   1:L PR[91] R[100]mm/sec CNT100;
   1:  PR[GP1:91,1] = PR[GP1:90,1] + -38.837;
   1:  PR[GP1:91,2] = PR[GP1:90,2] + -4.762;
   1:L PR[91] R[100]mm/sec CNT100;
   1:  PR[GP1:91,1] = PR[GP1:90,1] + -38.715;
   1:  PR[GP1:91,2] = PR[GP1:90,2] + -5.232;
   1:L PR[91] R[100]mm/sec CNT100;
   1:  PR[GP1:91,1] = PR[GP1:90,1] + -37.344;
   1:  PR[GP1:91,2] = PR[GP1:90,2] + -8.646;
   1:L PR[91] R[100]mm/sec CNT100;
   1:  PR[GP1:91,1] = PR[GP1:90,1] + -37.044;
   1:  PR[GP1:91,2] = PR[GP1:90,2] + -9.321;
   1:L PR[91] R[100]mm/sec CNT100;
   1:  PR[GP1:91,1] = PR[GP1:90,1] + -35.099;
   1:  PR[GP1:91,2] = PR[GP1:90,2] + -12.020;
   1:L PR[91] R[100]mm/sec CNT100;
   1:  PR[GP1:91,1] = PR[GP1:90,1] + -34.536;
   1:  PR[GP1:91,2] = PR[GP1:90,2] + -12.886;
   1:L PR[91] R[100]mm/sec CNT100;
   1:  PR[GP1:91,1] = PR[GP1:90,1] + -33.800;
   1:  PR[GP1:91,2] = PR[GP1:90,2] + -13.678;
   1:L PR[91] R[100]mm/sec CNT100;
   1:  PR[GP1:91,1] = PR[GP1:90,1] + -31.666;
   1:  PR[GP1:91,2] = PR[GP1:90,2] + -15.488;
   1:L PR[91] R[100]mm/sec CNT100;
   1:  PR[GP1:91,1] = PR[GP1:90,1] + -30.501;
   1:  PR[GP1:91,2] = PR[GP1:90,2] + -16.399;
   1:L PR[91] R[100]mm/sec CNT100;
   1:  PR[GP1:91,1] = PR[GP1:90,1] + -28.778;
   1:  PR[GP1:91,2] = PR[GP1:90,2] + -17.354;
   1:L PR[91] R[100]mm/sec CNT100;
   1:  PR[GP1:91,1] = PR[GP1:90,1] + -27.068;
   1:  PR[GP1:91,2] = PR[GP1:90,2] + -18.219;
   1:L PR[91] R[100]mm/sec CNT100;
   1:  PR[GP1:91,1] = PR[GP1:90,1] + -24.860;
   1:  PR[GP1:91,2] = PR[GP1:90,2] + -19.021;
   1:L PR[91] R[100]mm/sec CNT100;
   1:  PR[GP1:91,1] = PR[GP1:90,1] + -23.856;
   1:  PR[GP1:91,2] = PR[GP1:90,2] + -19.262;
   1:L PR[91] R[100]mm/sec CNT100;
   1:  PR[GP1:91,1] = PR[GP1:90,1] + -21.199;
   1:  PR[GP1:91,2] = PR[GP1:90,2] + -19.791;
   1:L PR[91] R[100]mm/sec CNT100;
   1:  PR[GP1:91,1] = PR[GP1:90,1] + -17.823;
   1:  PR[GP1:91,2] = PR[GP1:90,2] + -19.955;
   1:L PR[91] R[100]mm/sec CNT100;
   1:  PR[GP1:91,1] = PR[GP1:90,1] + -14.672;
   1:  PR[GP1:91,2] = PR[GP1:90,2] + -19.637;
   1:L PR[91] R[100]mm/sec CNT100;
   1:  PR[GP1:91,1] = PR[GP1:90,1] + -14.261;
   1:  PR[GP1:91,2] = PR[GP1:90,2] + -19.580;
   1:L PR[91] R[100]mm/sec CNT100;
   1:  PR[GP1:91,1] = PR[GP1:90,1] + -11.329;
   1:  PR[GP1:91,2] = PR[GP1:90,2] + -18.822;
   1:L PR[91] R[100]mm/sec CNT100;
   1:  PR[GP1:91,1] = PR[GP1:90,1] + -7.839;
   1:  PR[GP1:91,2] = PR[GP1:90,2] + -17.303;
   1:L PR[91] R[100]mm/sec CNT100;
   1:  PR[GP1:91,1] = PR[GP1:90,1] + -5.607;
   1:  PR[GP1:91,2] = PR[GP1:90,2] + -15.876;
   1:L PR[91] R[100]mm/sec CNT100;
   1:  PR[GP1:91,1] = PR[GP1:90,1] + -5.328;
   1:  PR[GP1:91,2] = PR[GP1:90,2] + -15.675;
   1:L PR[91] R[100]mm/sec CNT100;
   1:  PR[GP1:91,1] = PR[GP1:90,1] + -4.271;
   1:  PR[GP1:91,2] = PR[GP1:90,2] + -14.749;
   1:L PR[91] R[100]mm/sec CNT100;
   1:  PR[GP1:91,1] = PR[GP1:90,1] + -3.185;
   1:  PR[GP1:91,2] = PR[GP1:90,2] + -13.771;
   1:L PR[91] R[100]mm/sec CNT100;
   1:  PR[GP1:91,1] = PR[GP1:90,1] + -2.156;
   1:  PR[GP1:91,2] = PR[GP1:90,2] + -12.565;
   1:L PR[91] R[100]mm/sec CNT100;
   1:  PR[GP1:91,1] = PR[GP1:90,1] + -1.829;
   1:  PR[GP1:91,2] = PR[GP1:90,2] + -12.302;
   1:L PR[91] R[100]mm/sec CNT100;
   1:  PR[GP1:91,1] = PR[GP1:90,1] + -0.550;
   1:  PR[GP1:91,2] = PR[GP1:90,2] + -11.397;
   1:L PR[91] R[100]mm/sec CNT100;
   1:  PR[GP1:91,1] = PR[GP1:90,1] + 0.193;
   1:  PR[GP1:91,2] = PR[GP1:90,2] + -11.661;
   1:L PR[91] R[100]mm/sec CNT100;
   1:  PR[GP1:91,1] = PR[GP1:90,1] + 1.144;
   1:L PR[91] R[100]mm/sec CNT100;
   1:  PR[GP1:91,1] = PR[GP1:90,1] + 1.657;
   1:  PR[GP1:91,2] = PR[GP1:90,2] + -12.081;
   1:L PR[91] R[100]mm/sec CNT100;
   1:  PR[GP1:91,1] = PR[GP1:90,1] + 2.294;
   1:  PR[GP1:91,2] = PR[GP1:90,2] + -12.534;
   1:L PR[91] R[100]mm/sec CNT100;
   1:  PR[GP1:91,1] = PR[GP1:90,1] + 3.356;
   1:  PR[GP1:91,2] = PR[GP1:90,2] + -13.783;
   1:L PR[91] R[100]mm/sec CNT100;
   1:  PR[GP1:91,1] = PR[GP1:90,1] + 4.441;
   1:  PR[GP1:91,2] = PR[GP1:90,2] + -14.761;
   1:L PR[91] R[100]mm/sec CNT100;
   1:  PR[GP1:91,1] = PR[GP1:90,1] + 5.471;
   1:  PR[GP1:91,2] = PR[GP1:90,2] + -15.664;
   1:L PR[91] R[100]mm/sec CNT100;
   1:  PR[GP1:91,1] = PR[GP1:90,1] + 7.593;
   1:  PR[GP1:91,2] = PR[GP1:90,2] + -17.023;
   1:L PR[91] R[100]mm/sec CNT100;
   1:  PR[GP1:91,1] = PR[GP1:90,1] + 8.015;
   1:  PR[GP1:91,2] = PR[GP1:90,2] + -17.314;
   1:L PR[91] R[100]mm/sec CNT100;
   1:  PR[GP1:91,1] = PR[GP1:90,1] + 11.478;
   1:  PR[GP1:91,2] = PR[GP1:90,2] + -18.817;
   1:L PR[91] R[100]mm/sec CNT100;
   1:  PR[GP1:91,1] = PR[GP1:90,1] + 14.391;
   1:  PR[GP1:91,2] = PR[GP1:90,2] + -19.572;
   1:L PR[91] R[100]mm/sec CNT100;
   1:  PR[GP1:91,1] = PR[GP1:90,1] + 17.974;
   1:  PR[GP1:91,2] = PR[GP1:90,2] + -19.955;
   1:L PR[91] R[100]mm/sec CNT100;
   1:  PR[GP1:91,1] = PR[GP1:90,1] + 21.307;
   1:  PR[GP1:91,2] = PR[GP1:90,2] + -19.796;
   1:L PR[91] R[100]mm/sec CNT100;
   1:  PR[GP1:91,1] = PR[GP1:90,1] + 21.648;
   1:  PR[GP1:91,2] = PR[GP1:90,2] + -19.716;
   1:L PR[91] R[100]mm/sec CNT100;
   1:  PR[GP1:91,1] = PR[GP1:90,1] + 25.016;
   1:  PR[GP1:91,2] = PR[GP1:90,2] + -19.018;
   1:L PR[91] R[100]mm/sec CNT100;
   1:  PR[GP1:91,1] = PR[GP1:90,1] + 27.213;
   1:  PR[GP1:91,2] = PR[GP1:90,2] + -18.224;
   1:L PR[91] R[100]mm/sec CNT100;
   1:  PR[GP1:91,1] = PR[GP1:90,1] + 28.922;
   1:  PR[GP1:91,2] = PR[GP1:90,2] + -17.361;
   1:L PR[91] R[100]mm/sec CNT100;
   1:  PR[GP1:91,1] = PR[GP1:90,1] + 30.618;
   1:  PR[GP1:91,2] = PR[GP1:90,2] + -16.426;
   1:L PR[91] R[100]mm/sec CNT100;
   1:  PR[GP1:91,1] = PR[GP1:90,1] + 32.732;
   1:  PR[GP1:91,2] = PR[GP1:90,2] + -14.641;
   1:L PR[91] R[100]mm/sec CNT100;
   1:  PR[GP1:91,1] = PR[GP1:90,1] + 33.954;
   1:  PR[GP1:91,2] = PR[GP1:90,2] + -13.677;
   1:L PR[91] R[100]mm/sec CNT100;
   1:  PR[GP1:91,1] = PR[GP1:90,1] + 34.702;
   1:  PR[GP1:91,2] = PR[GP1:90,2] + -12.874;
   1:L PR[91] R[100]mm/sec CNT100;
   1:  PR[GP1:91,1] = PR[GP1:90,1] + 36.691;
   1:  PR[GP1:91,2] = PR[GP1:90,2] + -10.095;
   1:L PR[91] R[100]mm/sec CNT100;
   1:  PR[GP1:91,1] = PR[GP1:90,1] + 37.186;
   1:  PR[GP1:91,2] = PR[GP1:90,2] + -9.346;
   1:L PR[91] R[100]mm/sec CNT100;
   1:  PR[GP1:91,1] = PR[GP1:90,1] + 37.499;
   1:  PR[GP1:91,2] = PR[GP1:90,2] + -8.654;
   1:L PR[91] R[100]mm/sec CNT100;
   1:  PR[GP1:91,1] = PR[GP1:90,1] + 38.869;
   1:  PR[GP1:91,2] = PR[GP1:90,2] + -5.258;
   1:L PR[91] R[100]mm/sec CNT100;
   1:  PR[GP1:91,1] = PR[GP1:90,1] + 38.999;
   1:  PR[GP1:91,2] = PR[GP1:90,2] + -4.762;
   1:L PR[91] R[100]mm/sec CNT100;
   1:  PR[GP1:91,1] = PR[GP1:90,1] + 39.503;
   1:  PR[GP1:91,2] = PR[GP1:90,2] + -0.771;
   1:L PR[91] R[100]mm/sec CNT100;
   1:  PR[GP1:91,1] = PR[GP1:90,1] + 39.538;
   1:  PR[GP1:91,2] = PR[GP1:90,2] + -0.345;
   1:L PR[91] R[100]mm/sec CNT100;
   1:  PR[GP1:91,1] = PR[GP1:90,1] + 39.040;
   1:  PR[GP1:91,2] = PR[GP1:90,2] + 3.557;
   1:L PR[91] R[100]mm/sec CNT100;
   1:  PR[GP1:91,1] = PR[GP1:90,1] + 38.991;
   1:  PR[GP1:91,2] = PR[GP1:90,2] + 4.171;
   1:L PR[91] R[100]mm/sec CNT100;
   1:  PR[GP1:91,1] = PR[GP1:90,1] + 38.869;
   1:  PR[GP1:91,2] = PR[GP1:90,2] + 4.635;
   1:L PR[91] R[100]mm/sec CNT100;
   1:  PR[GP1:91,1] = PR[GP1:90,1] + 37.498;
   1:  PR[GP1:91,2] = PR[GP1:90,2] + 8.032;
   1:L PR[91] R[100]mm/sec CNT100;
   1:  PR[GP1:91,1] = PR[GP1:90,1] + 37.197;
   1:  PR[GP1:91,2] = PR[GP1:90,2] + 8.698;
   1:L PR[91] R[100]mm/sec CNT100;
   1:  PR[GP1:91,1] = PR[GP1:90,1] + 35.251;
   1:  PR[GP1:91,2] = PR[GP1:90,2] + 11.401;
   1:L PR[91] R[100]mm/sec CNT100;
   1:  PR[GP1:91,1] = PR[GP1:90,1] + 34.679;
   1:  PR[GP1:91,2] = PR[GP1:90,2] + 12.274;
   1:L PR[91] R[100]mm/sec CNT100;
   1:  PR[GP1:91,1] = PR[GP1:90,1] + 33.934;
   1:  PR[GP1:91,2] = PR[GP1:90,2] + 13.074;
   1:L PR[91] R[100]mm/sec CNT100;
   1:  PR[GP1:91,1] = PR[GP1:90,1] + 31.800;
   1:  PR[GP1:91,2] = PR[GP1:90,2] + 14.887;
   1:L PR[91] R[100]mm/sec CNT100;
   1:  PR[GP1:91,1] = PR[GP1:90,1] + 30.641;
   1:  PR[GP1:91,2] = PR[GP1:90,2] + 15.790;
   1:L PR[91] R[100]mm/sec CNT100;
   1:  PR[GP1:91,1] = PR[GP1:90,1] + 28.920;
   1:  PR[GP1:91,2] = PR[GP1:90,2] + 16.738;
   1:L PR[91] R[100]mm/sec CNT100;
   1:  PR[GP1:91,1] = PR[GP1:90,1] + 27.211;
   1:  PR[GP1:91,2] = PR[GP1:90,2] + 17.600;
   1:L PR[91] R[100]mm/sec CNT100;
   1:  PR[GP1:91,1] = PR[GP1:90,1] + 24.993;
   1:  PR[GP1:91,2] = PR[GP1:90,2] + 18.402;
   1:L PR[91] R[100]mm/sec CNT100;
   1:  PR[GP1:91,1] = PR[GP1:90,1] + 23.992;
   1:  PR[GP1:91,2] = PR[GP1:90,2] + 18.642;
   1:L PR[91] R[100]mm/sec CNT100;
   1:  PR[GP1:91,1] = PR[GP1:90,1] + 21.332;
   1:  PR[GP1:91,2] = PR[GP1:90,2] + 19.171;
   1:L PR[91] R[100]mm/sec CNT100;
   1:  PR[GP1:91,1] = PR[GP1:90,1] + 17.971;
   1:  PR[GP1:91,2] = PR[GP1:90,2] + 19.331;
   1:L PR[91] R[100]mm/sec CNT100;
   1:  PR[GP1:91,1] = PR[GP1:90,1] + 14.829;
   1:  PR[GP1:91,2] = PR[GP1:90,2] + 19.012;
   1:L PR[91] R[100]mm/sec CNT100;
   1:  PR[GP1:91,1] = PR[GP1:90,1] + 14.418;
   1:  PR[GP1:91,2] = PR[GP1:90,2] + 18.955;
   1:L PR[91] R[100]mm/sec CNT100;
   1:  PR[GP1:91,1] = PR[GP1:90,1] + 11.487;
   1:  PR[GP1:91,2] = PR[GP1:90,2] + 18.196;
   1:L PR[91] R[100]mm/sec CNT100;
   1:  PR[GP1:91,1] = PR[GP1:90,1] + 8.920;
   1:  PR[GP1:91,2] = PR[GP1:90,2] + 17.072;
   1:L PR[91] R[100]mm/sec CNT100;
   1:  PR[GP1:91,1] = PR[GP1:90,1] + 8.012;
   1:  PR[GP1:91,2] = PR[GP1:90,2] + 16.693;
   1:L PR[91] R[100]mm/sec CNT100;
   1:  PR[GP1:91,1] = PR[GP1:90,1] + 5.789;
   1:  PR[GP1:91,2] = PR[GP1:90,2] + 15.274;
   1:L PR[91] R[100]mm/sec CNT100;
   1:  PR[GP1:91,1] = PR[GP1:90,1] + 5.612;
   1:  PR[GP1:91,2] = PR[GP1:90,2] + 15.152;
   1:L PR[91] R[100]mm/sec CNT100;
   1:  PR[GP1:91,1] = PR[GP1:90,1] + 5.268;
   1:  PR[GP1:91,2] = PR[GP1:90,2] + 14.879;
   1:L PR[91] R[100]mm/sec CNT100;
   1:  PR[GP1:91,1] = PR[GP1:90,1] + 3.427;
   1:  PR[GP1:91,2] = PR[GP1:90,2] + 13.229;
   1:L PR[91] R[100]mm/sec CNT100;
   1:  PR[GP1:91,1] = PR[GP1:90,1] + 2.786;
   1:  PR[GP1:91,2] = PR[GP1:90,2] + 12.556;
   1:L PR[91] R[100]mm/sec CNT100;
   1:  PR[GP1:91,1] = PR[GP1:90,1] + 2.184;
   1:  PR[GP1:91,2] = PR[GP1:90,2] + 11.814;
   1:L PR[91] R[100]mm/sec CNT100;
   1:  PR[GP1:91,1] = PR[GP1:90,1] + 1.393;
   1:  PR[GP1:91,2] = PR[GP1:90,2] + 11.254;
   1:L PR[91] R[100]mm/sec CNT100;
   1:  PR[GP1:91,1] = PR[GP1:90,1] + 0.820;
   1:  PR[GP1:91,2] = PR[GP1:90,2] + 10.940;
   1:L PR[91] R[100]mm/sec CNT100;
   1:  PR[GP1:91,1] = PR[GP1:90,1] + -0.635;
   1:L PR[91] R[100]mm/sec CNT100;
   1:  PR[91] = PR[90];
   1:  PR[GP1:91,1] = PR[GP1:90,1] + -1.462;
   1:  PR[GP1:91,2] = PR[GP1:90,2] + 11.634;
   1:  PR[GP1:91,3] = PR[GP1:90,3] + 27.145;
   1:L PR[91] R[100]mm/sec CNT100;
   1:  PR[GP1:91,1] = PR[GP1:90,1] + -1.730;
   1:  PR[GP1:91,2] = PR[GP1:90,2] + 11.982;
   1:L PR[91] R[100]mm/sec CNT100;
   1:  PR[GP1:91,1] = PR[GP1:90,1] + -1.967;
   1:  PR[GP1:91,2] = PR[GP1:90,2] + 12.206;
   1:L PR[91] R[100]mm/sec CNT100;
   1:  PR[GP1:91,1] = PR[GP1:90,1] + -2.120;
   1:  PR[GP1:91,2] = PR[GP1:90,2] + 12.316;
   1:L PR[91] R[100]mm/sec CNT100;
   1:  PR[GP1:91,1] = PR[GP1:90,1] + -2.321;
   1:  PR[GP1:91,2] = PR[GP1:90,2] + 12.557;
   1:L PR[91] R[100]mm/sec CNT100;
   1:  PR[GP1:91,1] = PR[GP1:90,1] + -3.063;
   1:  PR[GP1:91,2] = PR[GP1:90,2] + 13.334;
   1:L PR[91] R[100]mm/sec CNT100;
   1:  PR[GP1:91,1] = PR[GP1:90,1] + -4.810;
   1:  PR[GP1:91,2] = PR[GP1:90,2] + 14.896;
   1:L PR[91] R[100]mm/sec CNT100;
   1:  PR[GP1:91,1] = PR[GP1:90,1] + -5.202;
   1:  PR[GP1:91,2] = PR[GP1:90,2] + 15.206;
   1:L PR[91] R[100]mm/sec CNT100;
   1:  PR[GP1:91,1] = PR[GP1:90,1] + -7.585;
   1:  PR[GP1:91,2] = PR[GP1:90,2] + 16.743;
   1:L PR[91] R[100]mm/sec CNT100;
   1:  PR[GP1:91,1] = PR[GP1:90,1] + -10.209;
   1:  PR[GP1:91,2] = PR[GP1:90,2] + 17.890;
   1:L PR[91] R[100]mm/sec CNT100;
   1:  PR[GP1:91,1] = PR[GP1:90,1] + -11.131;
   1:  PR[GP1:91,2] = PR[GP1:90,2] + 18.276;
   1:L PR[91] R[100]mm/sec CNT100;
   1:  PR[GP1:91,1] = PR[GP1:90,1] + -13.916;
   1:  PR[GP1:91,2] = PR[GP1:90,2] + 18.996;
   1:L PR[91] R[100]mm/sec CNT100;
   1:  PR[GP1:91,1] = PR[GP1:90,1] + -17.278;
   1:  PR[GP1:91,2] = PR[GP1:90,2] + 19.346;
   1:L PR[91] R[100]mm/sec CNT100;
   1:  PR[GP1:91,1] = PR[GP1:90,1] + -17.623;
   1:  PR[GP1:91,2] = PR[GP1:90,2] + 19.393;
   1:L PR[91] R[100]mm/sec CNT100;
   1:  PR[GP1:91,1] = PR[GP1:90,1] + -20.933;
   1:  PR[GP1:91,2] = PR[GP1:90,2] + 19.218;
   1:L PR[91] R[100]mm/sec CNT100;
   1:  PR[GP1:91,1] = PR[GP1:90,1] + -24.493;
   1:  PR[GP1:91,2] = PR[GP1:90,2] + 18.487;
   1:L PR[91] R[100]mm/sec CNT100;
   1:  PR[GP1:91,1] = PR[GP1:90,1] + -27.043;
   1:  PR[GP1:91,2] = PR[GP1:90,2] + 17.561;
   1:L PR[91] R[100]mm/sec CNT100;
   1:  PR[GP1:91,1] = PR[GP1:90,1] + -28.228;
   1:  PR[GP1:91,2] = PR[GP1:90,2] + 16.962;
   1:L PR[91] R[100]mm/sec CNT100;
   1:  PR[GP1:91,1] = PR[GP1:90,1] + -30.293;
   1:  PR[GP1:91,2] = PR[GP1:90,2] + 15.817;
   1:L PR[91] R[100]mm/sec CNT100;
   1:  PR[GP1:91,1] = PR[GP1:90,1] + -31.942;
   1:  PR[GP1:91,2] = PR[GP1:90,2] + 14.426;
   1:L PR[91] R[100]mm/sec CNT100;
   1:  PR[GP1:91,1] = PR[GP1:90,1] + -33.508;
   1:  PR[GP1:91,2] = PR[GP1:90,2] + 13.187;
   1:L PR[91] R[100]mm/sec CNT100;
   1:  PR[GP1:91,1] = PR[GP1:90,1] + -34.483;
   1:  PR[GP1:91,2] = PR[GP1:90,2] + 12.138;
   1:L PR[91] R[100]mm/sec CNT100;
   1:  PR[GP1:91,1] = PR[GP1:90,1] + -36.170;
   1:  PR[GP1:91,2] = PR[GP1:90,2] + 9.783;
   1:L PR[91] R[100]mm/sec CNT100;
   1:  PR[GP1:91,1] = PR[GP1:90,1] + -36.854;
   1:  PR[GP1:91,2] = PR[GP1:90,2] + 8.743;
   1:L PR[91] R[100]mm/sec CNT100;
   1:  PR[GP1:91,1] = PR[GP1:90,1] + -37.298;
   1:  PR[GP1:91,2] = PR[GP1:90,2] + 7.745;
   1:L PR[91] R[100]mm/sec CNT100;
   1:  PR[GP1:91,1] = PR[GP1:90,1] + -38.498;
   1:  PR[GP1:91,2] = PR[GP1:90,2] + 4.758;
   1:L PR[91] R[100]mm/sec CNT100;
   1:  PR[GP1:91,1] = PR[GP1:90,1] + -38.706;
   1:  PR[GP1:91,2] = PR[GP1:90,2] + 3.951;
   1:L PR[91] R[100]mm/sec CNT100;
   1:  PR[GP1:91,1] = PR[GP1:90,1] + -39.150;
   1:  PR[GP1:91,2] = PR[GP1:90,2] + 0.453;
   1:L PR[91] R[100]mm/sec CNT100;
   1:  PR[GP1:91,1] = PR[GP1:90,1] + -39.207;
   1:  PR[GP1:91,2] = PR[GP1:90,2] + -0.277;
   1:L PR[91] R[100]mm/sec CNT100;
   1:  PR[GP1:91,1] = PR[GP1:90,1] + -38.768;
   1:  PR[GP1:91,2] = PR[GP1:90,2] + -3.707;
   1:L PR[91] R[100]mm/sec CNT100;
   1:  PR[GP1:91,1] = PR[GP1:90,1] + -38.698;
   1:  PR[GP1:91,2] = PR[GP1:90,2] + -4.608;
   1:L PR[91] R[100]mm/sec CNT100;
   1:  PR[GP1:91,1] = PR[GP1:90,1] + -38.498;
   1:  PR[GP1:91,2] = PR[GP1:90,2] + -5.382;
   1:L PR[91] R[100]mm/sec CNT100;
   1:  PR[GP1:91,1] = PR[GP1:90,1] + -37.298;
   1:  PR[GP1:91,2] = PR[GP1:90,2] + -8.369;
   1:L PR[91] R[100]mm/sec CNT100;
   1:  PR[GP1:91,1] = PR[GP1:90,1] + -36.866;
   1:  PR[GP1:91,2] = PR[GP1:90,2] + -9.338;
   1:L PR[91] R[100]mm/sec CNT100;
   1:  PR[GP1:91,1] = PR[GP1:90,1] + -35.185;
   1:  PR[GP1:91,2] = PR[GP1:90,2] + -11.672;
   1:L PR[91] R[100]mm/sec CNT100;
   1:  PR[GP1:91,1] = PR[GP1:90,1] + -34.460;
   1:  PR[GP1:91,2] = PR[GP1:90,2] + -12.786;
   1:L PR[91] R[100]mm/sec CNT100;
   1:  PR[GP1:91,1] = PR[GP1:90,1] + -33.492;
   1:  PR[GP1:91,2] = PR[GP1:90,2] + -13.829;
   1:L PR[91] R[100]mm/sec CNT100;
   1:  PR[GP1:91,1] = PR[GP1:90,1] + -31.736;
   1:  PR[GP1:91,2] = PR[GP1:90,2] + -15.318;
   1:L PR[91] R[100]mm/sec CNT100;
   1:  PR[GP1:91,1] = PR[GP1:90,1] + -30.316;
   1:  PR[GP1:91,2] = PR[GP1:90,2] + -16.428;
   1:L PR[91] R[100]mm/sec CNT100;
   1:  PR[GP1:91,1] = PR[GP1:90,1] + -28.228;
   1:  PR[GP1:91,2] = PR[GP1:90,2] + -17.586;
   1:L PR[91] R[100]mm/sec CNT100;
   1:  PR[GP1:91,1] = PR[GP1:90,1] + -27.043;
   1:  PR[GP1:91,2] = PR[GP1:90,2] + -18.185;
   1:L PR[91] R[100]mm/sec CNT100;
   1:  PR[GP1:91,1] = PR[GP1:90,1] + -24.471;
   1:  PR[GP1:91,2] = PR[GP1:90,2] + -19.119;
   1:L PR[91] R[100]mm/sec CNT100;
   1:  PR[GP1:91,1] = PR[GP1:90,1] + -24.001;
   1:  PR[GP1:91,2] = PR[GP1:90,2] + -19.232;
   1:L PR[91] R[100]mm/sec CNT100;
   1:  PR[GP1:91,1] = PR[GP1:90,1] + -21.022;
   1:  PR[GP1:91,2] = PR[GP1:90,2] + -19.832;
   1:L PR[91] R[100]mm/sec CNT100;
   1:  PR[GP1:91,1] = PR[GP1:90,1] + -17.593;
   1:  PR[GP1:91,2] = PR[GP1:90,2] + -20.018;
   1:L PR[91] R[100]mm/sec CNT100;
   1:  PR[GP1:91,1] = PR[GP1:90,1] + -14.573;
   1:  PR[GP1:91,2] = PR[GP1:90,2] + -19.714;
   1:L PR[91] R[100]mm/sec CNT100;
   1:  PR[GP1:91,1] = PR[GP1:90,1] + -13.934;
   1:  PR[GP1:91,2] = PR[GP1:90,2] + -19.625;
   1:L PR[91] R[100]mm/sec CNT100;
   1:  PR[GP1:91,1] = PR[GP1:90,1] + -11.131;
   1:  PR[GP1:91,2] = PR[GP1:90,2] + -18.900;
   1:L PR[91] R[100]mm/sec CNT100;
   1:  PR[GP1:91,1] = PR[GP1:90,1] + -7.545;
   1:  PR[GP1:91,2] = PR[GP1:90,2] + -17.342;
   1:L PR[91] R[100]mm/sec CNT100;
   1:  PR[GP1:91,1] = PR[GP1:90,1] + -5.422;
   1:  PR[GP1:91,2] = PR[GP1:90,2] + -15.984;
   1:L PR[91] R[100]mm/sec CNT100;
   1:  PR[GP1:91,1] = PR[GP1:90,1] + -5.084;
   1:  PR[GP1:91,2] = PR[GP1:90,2] + -15.740;
   1:L PR[91] R[100]mm/sec CNT100;
   1:  PR[GP1:91,1] = PR[GP1:90,1] + -3.847;
   1:  PR[GP1:91,2] = PR[GP1:90,2] + -14.658;
   1:L PR[91] R[100]mm/sec CNT100;
   1:  PR[GP1:91,1] = PR[GP1:90,1] + -2.979;
   1:  PR[GP1:91,2] = PR[GP1:90,2] + -13.875;
   1:L PR[91] R[100]mm/sec CNT100;
   1:  PR[GP1:91,1] = PR[GP1:90,1] + -2.138;
   1:  PR[GP1:91,2] = PR[GP1:90,2] + -12.889;
   1:L PR[91] R[100]mm/sec CNT100;
   1:  PR[GP1:91,1] = PR[GP1:90,1] + -1.752;
   1:  PR[GP1:91,2] = PR[GP1:90,2] + -12.580;
   1:L PR[91] R[100]mm/sec CNT100;
   1:  PR[GP1:91,1] = PR[GP1:90,1] + -0.525;
   1:  PR[GP1:91,2] = PR[GP1:90,2] + -11.712;
   1:L PR[91] R[100]mm/sec CNT100;
   1:  PR[GP1:91,1] = PR[GP1:90,1] + 0.316;
   1:  PR[GP1:91,2] = PR[GP1:90,2] + -12.011;
   1:L PR[91] R[100]mm/sec CNT100;
   1:  PR[GP1:91,1] = PR[GP1:90,1] + 1.168;
   1:L PR[91] R[100]mm/sec CNT100;
   1:  PR[GP1:91,1] = PR[GP1:90,1] + 1.737;
   1:  PR[GP1:91,2] = PR[GP1:90,2] + -12.477;
   1:L PR[91] R[100]mm/sec CNT100;
   1:  PR[GP1:91,1] = PR[GP1:90,1] + 2.275;
   1:  PR[GP1:91,2] = PR[GP1:90,2] + -12.859;
   1:L PR[91] R[100]mm/sec CNT100;
   1:  PR[GP1:91,1] = PR[GP1:90,1] + 3.148;
   1:  PR[GP1:91,2] = PR[GP1:90,2] + -13.886;
   1:L PR[91] R[100]mm/sec CNT100;
   1:  PR[GP1:91,1] = PR[GP1:90,1] + 4.015;
   1:  PR[GP1:91,2] = PR[GP1:90,2] + -14.668;
   1:L PR[91] R[100]mm/sec CNT100;
   1:  PR[GP1:91,1] = PR[GP1:90,1] + 5.225;
   1:  PR[GP1:91,2] = PR[GP1:90,2] + -15.728;
   1:L PR[91] R[100]mm/sec CNT100;
   1:  PR[GP1:91,1] = PR[GP1:90,1] + 7.196;
   1:  PR[GP1:91,2] = PR[GP1:90,2] + -16.991;
   1:L PR[91] R[100]mm/sec CNT100;
   1:  PR[GP1:91,1] = PR[GP1:90,1] + 7.721;
   1:  PR[GP1:91,2] = PR[GP1:90,2] + -17.352;
   1:L PR[91] R[100]mm/sec CNT100;
   1:  PR[GP1:91,1] = PR[GP1:90,1] + 11.280;
   1:  PR[GP1:91,2] = PR[GP1:90,2] + -18.895;
   1:L PR[91] R[100]mm/sec CNT100;
   1:  PR[GP1:91,1] = PR[GP1:90,1] + 14.063;
   1:  PR[GP1:91,2] = PR[GP1:90,2] + -19.617;
   1:L PR[91] R[100]mm/sec CNT100;
   1:  PR[GP1:91,1] = PR[GP1:90,1] + 17.421;
   1:  PR[GP1:91,2] = PR[GP1:90,2] + -19.969;
   1:L PR[91] R[100]mm/sec CNT100;
   1:  PR[GP1:91,1] = PR[GP1:90,1] + 17.768;
   1:  PR[GP1:91,2] = PR[GP1:90,2] + -20.017;
   1:L PR[91] R[100]mm/sec CNT100;
   1:  PR[GP1:91,1] = PR[GP1:90,1] + 21.063;
   1:  PR[GP1:91,2] = PR[GP1:90,2] + -19.846;
   1:L PR[91] R[100]mm/sec CNT100;
   1:  PR[GP1:91,1] = PR[GP1:90,1] + 24.625;
   1:  PR[GP1:91,2] = PR[GP1:90,2] + -19.116;
   1:L PR[91] R[100]mm/sec CNT100;
   1:  PR[GP1:91,1] = PR[GP1:90,1] + 27.186;
   1:  PR[GP1:91,2] = PR[GP1:90,2] + -18.191;
   1:L PR[91] R[100]mm/sec CNT100;
   1:  PR[GP1:91,1] = PR[GP1:90,1] + 28.369;
   1:  PR[GP1:91,2] = PR[GP1:90,2] + -17.594;
   1:L PR[91] R[100]mm/sec CNT100;
   1:  PR[GP1:91,1] = PR[GP1:90,1] + 30.431;
   1:  PR[GP1:91,2] = PR[GP1:90,2] + -16.457;
   1:L PR[91] R[100]mm/sec CNT100;
   1:  PR[GP1:91,1] = PR[GP1:90,1] + 32.078;
   1:  PR[GP1:91,2] = PR[GP1:90,2] + -15.066;
   1:L PR[91] R[100]mm/sec CNT100;
   1:  PR[GP1:91,1] = PR[GP1:90,1] + 33.640;
   1:  PR[GP1:91,2] = PR[GP1:90,2] + -13.833;
   1:L PR[91] R[100]mm/sec CNT100;
   1:  PR[GP1:91,1] = PR[GP1:90,1] + 34.622;
   1:  PR[GP1:91,2] = PR[GP1:90,2] + -12.778;
   1:L PR[91] R[100]mm/sec CNT100;
   1:  PR[GP1:91,1] = PR[GP1:90,1] + 36.310;
   1:  PR[GP1:91,2] = PR[GP1:90,2] + -10.421;
   1:L PR[91] R[100]mm/sec CNT100;
   1:  PR[GP1:91,1] = PR[GP1:90,1] + 37.008;
   1:  PR[GP1:91,2] = PR[GP1:90,2] + -9.366;
   1:L PR[91] R[100]mm/sec CNT100;
   1:  PR[GP1:91,1] = PR[GP1:90,1] + 37.451;
   1:  PR[GP1:91,2] = PR[GP1:90,2] + -8.384;
   1:L PR[91] R[100]mm/sec CNT100;
   1:  PR[GP1:91,1] = PR[GP1:90,1] + 38.650;
   1:  PR[GP1:91,2] = PR[GP1:90,2] + -5.412;
   1:L PR[91] R[100]mm/sec CNT100;
   1:  PR[GP1:91,1] = PR[GP1:90,1] + 38.859;
   1:  PR[GP1:91,2] = PR[GP1:90,2] + -4.616;
   1:L PR[91] R[100]mm/sec CNT100;
   1:  PR[GP1:91,1] = PR[GP1:90,1] + 39.303;
   1:  PR[GP1:91,2] = PR[GP1:90,2] + -1.104;
   1:L PR[91] R[100]mm/sec CNT100;
   1:  PR[GP1:91,1] = PR[GP1:90,1] + 39.364;
   1:  PR[GP1:91,2] = PR[GP1:90,2] + -0.345;
   1:L PR[91] R[100]mm/sec CNT100;
   1:  PR[GP1:91,1] = PR[GP1:90,1] + 38.925;
   1:  PR[GP1:91,2] = PR[GP1:90,2] + 3.096;
   1:L PR[91] R[100]mm/sec CNT100;
   1:  PR[GP1:91,1] = PR[GP1:90,1] + 38.850;
   1:  PR[GP1:91,2] = PR[GP1:90,2] + 4.025;
   1:L PR[91] R[100]mm/sec CNT100;
   1:  PR[GP1:91,1] = PR[GP1:90,1] + 38.650;
   1:  PR[GP1:91,2] = PR[GP1:90,2] + 4.789;
   1:L PR[91] R[100]mm/sec CNT100;
   1:  PR[GP1:91,1] = PR[GP1:90,1] + 37.450;
   1:  PR[GP1:91,2] = PR[GP1:90,2] + 7.761;
   1:L PR[91] R[100]mm/sec CNT100;
   1:  PR[GP1:91,1] = PR[GP1:90,1] + 37.019;
   1:  PR[GP1:91,2] = PR[GP1:90,2] + 8.717;
   1:L PR[91] R[100]mm/sec CNT100;
   1:  PR[GP1:91,1] = PR[GP1:90,1] + 35.335;
   1:  PR[GP1:91,2] = PR[GP1:90,2] + 11.055;
   1:L PR[91] R[100]mm/sec CNT100;
   1:  PR[GP1:91,1] = PR[GP1:90,1] + 34.600;
   1:  PR[GP1:91,2] = PR[GP1:90,2] + 12.178;
   1:L PR[91] R[100]mm/sec CNT100;
   1:  PR[GP1:91,1] = PR[GP1:90,1] + 33.621;
   1:  PR[GP1:91,2] = PR[GP1:90,2] + 13.230;
   1:L PR[91] R[100]mm/sec CNT100;
   1:  PR[GP1:91,1] = PR[GP1:90,1] + 31.866;
   1:  PR[GP1:91,2] = PR[GP1:90,2] + 14.721;
   1:L PR[91] R[100]mm/sec CNT100;
   1:  PR[GP1:91,1] = PR[GP1:90,1] + 30.454;
   1:  PR[GP1:91,2] = PR[GP1:90,2] + 15.820;
   1:L PR[91] R[100]mm/sec CNT100;
   1:  PR[GP1:91,1] = PR[GP1:90,1] + 28.367;
   1:  PR[GP1:91,2] = PR[GP1:90,2] + 16.971;
   1:L PR[91] R[100]mm/sec CNT100;
   1:  PR[GP1:91,1] = PR[GP1:90,1] + 27.184;
   1:  PR[GP1:91,2] = PR[GP1:90,2] + 17.567;
   1:L PR[91] R[100]mm/sec CNT100;
   1:  PR[GP1:91,1] = PR[GP1:90,1] + 24.601;
   1:  PR[GP1:91,2] = PR[GP1:90,2] + 18.501;
   1:L PR[91] R[100]mm/sec CNT100;
   1:  PR[GP1:91,1] = PR[GP1:90,1] + 24.135;
   1:  PR[GP1:91,2] = PR[GP1:90,2] + 18.613;
   1:L PR[91] R[100]mm/sec CNT100;
   1:  PR[GP1:91,1] = PR[GP1:90,1] + 21.156;
   1:  PR[GP1:91,2] = PR[GP1:90,2] + 19.212;
   1:L PR[91] R[100]mm/sec CNT100;
   1:  PR[GP1:91,1] = PR[GP1:90,1] + 17.743;
   1:  PR[GP1:91,2] = PR[GP1:90,2] + 19.395;
   1:L PR[91] R[100]mm/sec CNT100;
   1:  PR[GP1:91,1] = PR[GP1:90,1] + 14.732;
   1:  PR[GP1:91,2] = PR[GP1:90,2] + 19.089;
   1:L PR[91] R[100]mm/sec CNT100;
   1:  PR[GP1:91,1] = PR[GP1:90,1] + 14.093;
   1:  PR[GP1:91,2] = PR[GP1:90,2] + 19.001;
   1:L PR[91] R[100]mm/sec CNT100;
   1:  PR[GP1:91,1] = PR[GP1:90,1] + 11.291;
   1:  PR[GP1:91,2] = PR[GP1:90,2] + 18.274;
   1:L PR[91] R[100]mm/sec CNT100;
   1:  PR[GP1:91,1] = PR[GP1:90,1] + 8.834;
   1:  PR[GP1:91,2] = PR[GP1:90,2] + 17.199;
   1:L PR[91] R[100]mm/sec CNT100;
   1:  PR[GP1:91,1] = PR[GP1:90,1] + 7.725;
   1:  PR[GP1:91,2] = PR[GP1:90,2] + 16.736;
   1:L PR[91] R[100]mm/sec CNT100;
   1:  PR[GP1:91,1] = PR[GP1:90,1] + 5.607;
   1:  PR[GP1:91,2] = PR[GP1:90,2] + 15.384;
   1:L PR[91] R[100]mm/sec CNT100;
   1:  PR[GP1:91,1] = PR[GP1:90,1] + 5.391;
   1:  PR[GP1:91,2] = PR[GP1:90,2] + 15.235;
   1:L PR[91] R[100]mm/sec CNT100;
   1:  PR[GP1:91,1] = PR[GP1:90,1] + 4.980;
   1:  PR[GP1:91,2] = PR[GP1:90,2] + 14.909;
   1:L PR[91] R[100]mm/sec CNT100;
   1:  PR[GP1:91,1] = PR[GP1:90,1] + 3.232;
   1:  PR[GP1:91,2] = PR[GP1:90,2] + 13.345;
   1:L PR[91] R[100]mm/sec CNT100;
   1:  PR[GP1:91,1] = PR[GP1:90,1] + 2.501;
   1:  PR[GP1:91,2] = PR[GP1:90,2] + 12.576;
   1:L PR[91] R[100]mm/sec CNT100;
   1:  PR[GP1:91,1] = PR[GP1:90,1] + 2.136;
   1:  PR[GP1:91,2] = PR[GP1:90,2] + 12.113;
   1:L PR[91] R[100]mm/sec CNT100;
   1:  PR[GP1:91,1] = PR[GP1:90,1] + 1.418;
   1:  PR[GP1:91,2] = PR[GP1:90,2] + 11.604;
   1:L PR[91] R[100]mm/sec CNT100;
   1:  PR[GP1:91,1] = PR[GP1:90,1] + 0.780;
   1:  PR[GP1:91,2] = PR[GP1:90,2] + 11.255;
   1:L PR[91] R[100]mm/sec CNT100;
   1:  PR[GP1:91,1] = PR[GP1:90,1] + -0.611;
   1:L PR[91] R[100]mm/sec CNT100;
   1:  PR[91] = PR[90];
   1:  PR[GP1:91,1] = PR[GP1:90,1] + -1.502;
   1:  PR[GP1:91,2] = PR[GP1:90,2] + 11.977;
   1:  PR[GP1:91,3] = PR[GP1:90,3] + 27.755;
   1:L PR[91] R[100]mm/sec CNT100;
   1:  PR[GP1:91,1] = PR[GP1:90,1] + -1.800;
   1:  PR[GP1:91,2] = PR[GP1:90,2] + 12.366;
   1:L PR[91] R[100]mm/sec CNT100;
   1:  PR[GP1:91,1] = PR[GP1:90,1] + -2.127;
   1:  PR[GP1:91,2] = PR[GP1:90,2] + 12.673;
   1:L PR[91] R[100]mm/sec CNT100;
   1:  PR[GP1:91,1] = PR[GP1:90,1] + -2.870;
   1:  PR[GP1:91,2] = PR[GP1:90,2] + 13.451;
   1:L PR[91] R[100]mm/sec CNT100;
   1:  PR[GP1:91,1] = PR[GP1:90,1] + -4.523;
   1:  PR[GP1:91,2] = PR[GP1:90,2] + 14.927;
   1:L PR[91] R[100]mm/sec CNT100;
   1:  PR[GP1:91,1] = PR[GP1:90,1] + -4.983;
   1:  PR[GP1:91,2] = PR[GP1:90,2] + 15.290;
   1:L PR[91] R[100]mm/sec CNT100;
   1:  PR[GP1:91,1] = PR[GP1:90,1] + -7.298;
   1:  PR[GP1:91,2] = PR[GP1:90,2] + 16.786;
   1:L PR[91] R[100]mm/sec CNT100;
   1:  PR[GP1:91,1] = PR[GP1:90,1] + -9.793;
   1:  PR[GP1:91,2] = PR[GP1:90,2] + 17.877;
   1:L PR[91] R[100]mm/sec CNT100;
   1:  PR[GP1:91,1] = PR[GP1:90,1] + -10.935;
   1:  PR[GP1:91,2] = PR[GP1:90,2] + 18.355;
   1:L PR[91] R[100]mm/sec CNT100;
   1:  PR[GP1:91,1] = PR[GP1:90,1] + -13.591;
   1:  PR[GP1:91,2] = PR[GP1:90,2] + 19.042;
   1:L PR[91] R[100]mm/sec CNT100;
   1:  PR[GP1:91,1] = PR[GP1:90,1] + -16.804;
   1:  PR[GP1:91,2] = PR[GP1:90,2] + 19.376;
   1:L PR[91] R[100]mm/sec CNT100;
   1:  PR[GP1:91,1] = PR[GP1:90,1] + -17.398;
   1:  PR[GP1:91,2] = PR[GP1:90,2] + 19.457;
   1:L PR[91] R[100]mm/sec CNT100;
   1:  PR[GP1:91,1] = PR[GP1:90,1] + -20.627;
   1:  PR[GP1:91,2] = PR[GP1:90,2] + 19.287;
   1:L PR[91] R[100]mm/sec CNT100;
   1:  PR[GP1:91,1] = PR[GP1:90,1] + -20.849;
   1:  PR[GP1:91,2] = PR[GP1:90,2] + 19.261;
   1:L PR[91] R[100]mm/sec CNT100;
   1:  PR[GP1:91,1] = PR[GP1:90,1] + -24.103;
   1:  PR[GP1:91,2] = PR[GP1:90,2] + 18.585;
   1:L PR[91] R[100]mm/sec CNT100;
   1:  PR[GP1:91,1] = PR[GP1:90,1] + -27.017;
   1:  PR[GP1:91,2] = PR[GP1:90,2] + 17.527;
   1:L PR[91] R[100]mm/sec CNT100;
   1:  PR[GP1:91,1] = PR[GP1:90,1] + -27.677;
   1:  PR[GP1:91,2] = PR[GP1:90,2] + 17.193;
   1:L PR[91] R[100]mm/sec CNT100;
   1:  PR[GP1:91,1] = PR[GP1:90,1] + -30.109;
   1:  PR[GP1:91,2] = PR[GP1:90,2] + 15.845;
   1:L PR[91] R[100]mm/sec CNT100;
   1:  PR[GP1:91,1] = PR[GP1:90,1] + -31.292;
   1:  PR[GP1:91,2] = PR[GP1:90,2] + 14.847;
   1:L PR[91] R[100]mm/sec CNT100;
   1:  PR[GP1:91,1] = PR[GP1:90,1] + -33.200;
   1:  PR[GP1:91,2] = PR[GP1:90,2] + 13.337;
   1:L PR[91] R[100]mm/sec CNT100;
   1:  PR[GP1:91,1] = PR[GP1:90,1] + -34.407;
   1:  PR[GP1:91,2] = PR[GP1:90,2] + 12.039;
   1:L PR[91] R[100]mm/sec CNT100;
   1:  PR[GP1:91,1] = PR[GP1:90,1] + -35.794;
   1:  PR[GP1:91,2] = PR[GP1:90,2] + 10.103;
   1:L PR[91] R[100]mm/sec CNT100;
   1:  PR[GP1:91,1] = PR[GP1:90,1] + -36.677;
   1:  PR[GP1:91,2] = PR[GP1:90,2] + 8.760;
   1:L PR[91] R[100]mm/sec CNT100;
   1:  PR[GP1:91,1] = PR[GP1:90,1] + -37.252;
   1:  PR[GP1:91,2] = PR[GP1:90,2] + 7.468;
   1:L PR[91] R[100]mm/sec CNT100;
   1:  PR[GP1:91,1] = PR[GP1:90,1] + -38.280;
   1:  PR[GP1:91,2] = PR[GP1:90,2] + 4.908;
   1:L PR[91] R[100]mm/sec CNT100;
   1:  PR[GP1:91,1] = PR[GP1:90,1] + -38.567;
   1:  PR[GP1:91,2] = PR[GP1:90,2] + 3.797;
   1:L PR[91] R[100]mm/sec CNT100;
   1:  PR[GP1:91,1] = PR[GP1:90,1] + -38.950;
   1:  PR[GP1:91,2] = PR[GP1:90,2] + 0.776;
   1:L PR[91] R[100]mm/sec CNT100;
   1:  PR[GP1:91,1] = PR[GP1:90,1] + -39.033;
   1:  PR[GP1:91,2] = PR[GP1:90,2] + -0.277;
   1:L PR[91] R[100]mm/sec CNT100;
   1:  PR[GP1:91,1] = PR[GP1:90,1] + -38.653;
   1:  PR[GP1:91,2] = PR[GP1:90,2] + -3.247;
   1:L PR[91] R[100]mm/sec CNT100;
   1:  PR[GP1:91,1] = PR[GP1:90,1] + -38.559;
   1:  PR[GP1:91,2] = PR[GP1:90,2] + -4.454;
   1:L PR[91] R[100]mm/sec CNT100;
   1:  PR[GP1:91,1] = PR[GP1:90,1] + -38.280;
   1:  PR[GP1:91,2] = PR[GP1:90,2] + -5.532;
   1:L PR[91] R[100]mm/sec CNT100;
   1:  PR[GP1:91,1] = PR[GP1:90,1] + -37.252;
   1:  PR[GP1:91,2] = PR[GP1:90,2] + -8.092;
   1:L PR[91] R[100]mm/sec CNT100;
   1:  PR[GP1:91,1] = PR[GP1:90,1] + -36.689;
   1:  PR[GP1:91,2] = PR[GP1:90,2] + -9.355;
   1:L PR[91] R[100]mm/sec CNT100;
   1:  PR[GP1:91,1] = PR[GP1:90,1] + -35.270;
   1:  PR[GP1:91,2] = PR[GP1:90,2] + -11.324;
   1:L PR[91] R[100]mm/sec CNT100;
   1:  PR[GP1:91,1] = PR[GP1:90,1] + -34.385;
   1:  PR[GP1:91,2] = PR[GP1:90,2] + -12.687;
   1:L PR[91] R[100]mm/sec CNT100;
   1:  PR[GP1:91,1] = PR[GP1:90,1] + -33.183;
   1:  PR[GP1:91,2] = PR[GP1:90,2] + -13.979;
   1:L PR[91] R[100]mm/sec CNT100;
   1:  PR[GP1:91,1] = PR[GP1:90,1] + -31.805;
   1:  PR[GP1:91,2] = PR[GP1:90,2] + -15.148;
   1:L PR[91] R[100]mm/sec CNT100;
   1:  PR[GP1:91,1] = PR[GP1:90,1] + -30.132;
   1:  PR[GP1:91,2] = PR[GP1:90,2] + -16.456;
   1:L PR[91] R[100]mm/sec CNT100;
   1:  PR[GP1:91,1] = PR[GP1:90,1] + -27.677;
   1:  PR[GP1:91,2] = PR[GP1:90,2] + -17.817;
   1:L PR[91] R[100]mm/sec CNT100;
   1:  PR[GP1:91,1] = PR[GP1:90,1] + -27.017;
   1:  PR[GP1:91,2] = PR[GP1:90,2] + -18.151;
   1:L PR[91] R[100]mm/sec CNT100;
   1:  PR[GP1:91,1] = PR[GP1:90,1] + -24.103;
   1:  PR[GP1:91,2] = PR[GP1:90,2] + -19.209;
   1:L PR[91] R[100]mm/sec CNT100;
   1:  PR[GP1:91,1] = PR[GP1:90,1] + -20.848;
   1:  PR[GP1:91,2] = PR[GP1:90,2] + -19.885;
   1:L PR[91] R[100]mm/sec CNT100;
   1:  PR[GP1:91,1] = PR[GP1:90,1] + -20.625;
   1:  PR[GP1:91,2] = PR[GP1:90,2] + -19.911;
   1:L PR[91] R[100]mm/sec CNT100;
   1:  PR[GP1:91,1] = PR[GP1:90,1] + -17.368;
   1:  PR[GP1:91,2] = PR[GP1:90,2] + -20.082;
   1:L PR[91] R[100]mm/sec CNT100;
   1:  PR[GP1:91,1] = PR[GP1:90,1] + -14.474;
   1:  PR[GP1:91,2] = PR[GP1:90,2] + -19.791;
   1:L PR[91] R[100]mm/sec CNT100;
   1:  PR[GP1:91,1] = PR[GP1:90,1] + -13.607;
   1:  PR[GP1:91,2] = PR[GP1:90,2] + -19.670;
   1:L PR[91] R[100]mm/sec CNT100;
   1:  PR[GP1:91,1] = PR[GP1:90,1] + -10.936;
   1:  PR[GP1:91,2] = PR[GP1:90,2] + -18.979;
   1:L PR[91] R[100]mm/sec CNT100;
   1:  PR[GP1:91,1] = PR[GP1:90,1] + -8.588;
   1:  PR[GP1:91,2] = PR[GP1:90,2] + -17.949;
   1:L PR[91] R[100]mm/sec CNT100;
   1:  PR[GP1:91,1] = PR[GP1:90,1] + -7.248;
   1:  PR[GP1:91,2] = PR[GP1:90,2] + -17.378;
   1:L PR[91] R[100]mm/sec CNT100;
   1:  PR[GP1:91,1] = PR[GP1:90,1] + -5.237;
   1:  PR[GP1:91,2] = PR[GP1:90,2] + -16.092;
   1:L PR[91] R[100]mm/sec CNT100;
   1:  PR[GP1:91,1] = PR[GP1:90,1] + -4.843;
   1:  PR[GP1:91,2] = PR[GP1:90,2] + -15.808;
   1:L PR[91] R[100]mm/sec CNT100;
   1:  PR[GP1:91,1] = PR[GP1:90,1] + -2.769;
   1:  PR[GP1:91,2] = PR[GP1:90,2] + -13.975;
   1:L PR[91] R[100]mm/sec CNT100;
   1:  PR[GP1:91,1] = PR[GP1:90,1] + -2.120;
   1:  PR[GP1:91,2] = PR[GP1:90,2] + -13.214;
   1:L PR[91] R[100]mm/sec CNT100;
   1:  PR[GP1:91,1] = PR[GP1:90,1] + -1.676;
   1:  PR[GP1:91,2] = PR[GP1:90,2] + -12.857;
   1:L PR[91] R[100]mm/sec CNT100;
   1:  PR[GP1:91,1] = PR[GP1:90,1] + -0.501;
   1:  PR[GP1:91,2] = PR[GP1:90,2] + -12.027;
   1:L PR[91] R[100]mm/sec CNT100;
   1:  PR[GP1:91,1] = PR[GP1:90,1] + 0.440;
   1:  PR[GP1:91,2] = PR[GP1:90,2] + -12.361;
   1:L PR[91] R[100]mm/sec CNT100;
   1:  PR[GP1:91,1] = PR[GP1:90,1] + 1.193;
   1:L PR[91] R[100]mm/sec CNT100;
   1:  PR[GP1:91,1] = PR[GP1:90,1] + 1.817;
   1:  PR[GP1:91,2] = PR[GP1:90,2] + -12.872;
   1:L PR[91] R[100]mm/sec CNT100;
   1:  PR[GP1:91,1] = PR[GP1:90,1] + 2.256;
   1:  PR[GP1:91,2] = PR[GP1:90,2] + -13.184;
   1:L PR[91] R[100]mm/sec CNT100;
   1:  PR[GP1:91,1] = PR[GP1:90,1] + 2.936;
   1:  PR[GP1:91,2] = PR[GP1:90,2] + -13.984;
   1:L PR[91] R[100]mm/sec CNT100;
   1:  PR[GP1:91,1] = PR[GP1:90,1] + 4.982;
   1:  PR[GP1:91,2] = PR[GP1:90,2] + -15.795;
   1:L PR[91] R[100]mm/sec CNT100;
   1:  PR[GP1:91,1] = PR[GP1:90,1] + 6.799;
   1:  PR[GP1:91,2] = PR[GP1:90,2] + -16.959;
   1:L PR[91] R[100]mm/sec CNT100;
   1:  PR[GP1:91,1] = PR[GP1:90,1] + 7.427;
   1:  PR[GP1:91,2] = PR[GP1:90,2] + -17.391;
   1:L PR[91] R[100]mm/sec CNT100;
   1:  PR[GP1:91,1] = PR[GP1:90,1] + 11.082;
   1:  PR[GP1:91,2] = PR[GP1:90,2] + -18.974;
   1:L PR[91] R[100]mm/sec CNT100;
   1:  PR[GP1:91,1] = PR[GP1:90,1] + 13.736;
   1:  PR[GP1:91,2] = PR[GP1:90,2] + -19.662;
   1:L PR[91] R[100]mm/sec CNT100;
   1:  PR[GP1:91,1] = PR[GP1:90,1] + 16.945;
   1:  PR[GP1:91,2] = PR[GP1:90,2] + -19.998;
   1:L PR[91] R[100]mm/sec CNT100;
   1:  PR[GP1:91,1] = PR[GP1:90,1] + 17.542;
   1:  PR[GP1:91,2] = PR[GP1:90,2] + -20.081;
   1:L PR[91] R[100]mm/sec CNT100;
   1:  PR[GP1:91,1] = PR[GP1:90,1] + 20.757;
   1:  PR[GP1:91,2] = PR[GP1:90,2] + -19.914;
   1:L PR[91] R[100]mm/sec CNT100;
   1:  PR[GP1:91,1] = PR[GP1:90,1] + 20.981;
   1:  PR[GP1:91,2] = PR[GP1:90,2] + -19.888;
   1:L PR[91] R[100]mm/sec CNT100;
   1:  PR[GP1:91,1] = PR[GP1:90,1] + 24.231;
   1:  PR[GP1:91,2] = PR[GP1:90,2] + -19.216;
   1:L PR[91] R[100]mm/sec CNT100;
   1:  PR[GP1:91,1] = PR[GP1:90,1] + 27.158;
   1:  PR[GP1:91,2] = PR[GP1:90,2] + -18.158;
   1:L PR[91] R[100]mm/sec CNT100;
   1:  PR[GP1:91,1] = PR[GP1:90,1] + 27.815;
   1:  PR[GP1:91,2] = PR[GP1:90,2] + -17.826;
   1:L PR[91] R[100]mm/sec CNT100;
   1:  PR[GP1:91,1] = PR[GP1:90,1] + 30.243;
   1:  PR[GP1:91,2] = PR[GP1:90,2] + -16.487;
   1:L PR[91] R[100]mm/sec CNT100;
   1:  PR[GP1:91,1] = PR[GP1:90,1] + 31.424;
   1:  PR[GP1:91,2] = PR[GP1:90,2] + -15.490;
   1:L PR[91] R[100]mm/sec CNT100;
   1:  PR[GP1:91,1] = PR[GP1:90,1] + 33.327;
   1:  PR[GP1:91,2] = PR[GP1:90,2] + -13.989;
   1:L PR[91] R[100]mm/sec CNT100;
   1:  PR[GP1:91,1] = PR[GP1:90,1] + 34.543;
   1:  PR[GP1:91,2] = PR[GP1:90,2] + -12.683;
   1:L PR[91] R[100]mm/sec CNT100;
   1:  PR[GP1:91,1] = PR[GP1:90,1] + 35.930;
   1:  PR[GP1:91,2] = PR[GP1:90,2] + -10.746;
   1:L PR[91] R[100]mm/sec CNT100;
   1:  PR[GP1:91,1] = PR[GP1:90,1] + 36.829;
   1:  PR[GP1:91,2] = PR[GP1:90,2] + -9.386;
   1:L PR[91] R[100]mm/sec CNT100;
   1:  PR[GP1:91,1] = PR[GP1:90,1] + 37.404;
   1:  PR[GP1:91,2] = PR[GP1:90,2] + -8.113;
   1:L PR[91] R[100]mm/sec CNT100;
   1:  PR[GP1:91,1] = PR[GP1:90,1] + 38.431;
   1:  PR[GP1:91,2] = PR[GP1:90,2] + -5.567;
   1:L PR[91] R[100]mm/sec CNT100;
   1:  PR[GP1:91,1] = PR[GP1:90,1] + 38.718;
   1:  PR[GP1:91,2] = PR[GP1:90,2] + -4.469;
   1:L PR[91] R[100]mm/sec CNT100;
   1:  PR[GP1:91,1] = PR[GP1:90,1] + 39.102;
   1:  PR[GP1:91,2] = PR[GP1:90,2] + -1.437;
   1:L PR[91] R[100]mm/sec CNT100;
   1:  PR[GP1:91,1] = PR[GP1:90,1] + 39.190;
   1:  PR[GP1:91,2] = PR[GP1:90,2] + -0.345;
   1:L PR[91] R[100]mm/sec CNT100;
   1:  PR[GP1:91,1] = PR[GP1:90,1] + 38.810;
   1:  PR[GP1:91,2] = PR[GP1:90,2] + 2.635;
   1:L PR[91] R[100]mm/sec CNT100;
   1:  PR[GP1:91,1] = PR[GP1:90,1] + 38.710;
   1:  PR[GP1:91,2] = PR[GP1:90,2] + 3.878;
   1:L PR[91] R[100]mm/sec CNT100;
   1:  PR[GP1:91,1] = PR[GP1:90,1] + 38.430;
   1:  PR[GP1:91,2] = PR[GP1:90,2] + 4.944;
   1:L PR[91] R[100]mm/sec CNT100;
   1:  PR[GP1:91,1] = PR[GP1:90,1] + 37.403;
   1:  PR[GP1:91,2] = PR[GP1:90,2] + 7.490;
   1:L PR[91] R[100]mm/sec CNT100;
   1:  PR[GP1:91,1] = PR[GP1:90,1] + 36.840;
   1:  PR[GP1:91,2] = PR[GP1:90,2] + 8.736;
   1:L PR[91] R[100]mm/sec CNT100;
   1:  PR[GP1:91,1] = PR[GP1:90,1] + 35.420;
   1:  PR[GP1:91,2] = PR[GP1:90,2] + 10.708;
   1:L PR[91] R[100]mm/sec CNT100;
   1:  PR[GP1:91,1] = PR[GP1:90,1] + 34.521;
   1:  PR[GP1:91,2] = PR[GP1:90,2] + 12.083;
   1:L PR[91] R[100]mm/sec CNT100;
   1:  PR[GP1:91,1] = PR[GP1:90,1] + 33.307;
   1:  PR[GP1:91,2] = PR[GP1:90,2] + 13.386;
   1:L PR[91] R[100]mm/sec CNT100;
   1:  PR[GP1:91,1] = PR[GP1:90,1] + 31.932;
   1:  PR[GP1:91,2] = PR[GP1:90,2] + 14.555;
   1:L PR[91] R[100]mm/sec CNT100;
   1:  PR[GP1:91,1] = PR[GP1:90,1] + 30.267;
   1:  PR[GP1:91,2] = PR[GP1:90,2] + 15.850;
   1:L PR[91] R[100]mm/sec CNT100;
   1:  PR[GP1:91,1] = PR[GP1:90,1] + 27.814;
   1:  PR[GP1:91,2] = PR[GP1:90,2] + 17.202;
   1:L PR[91] R[100]mm/sec CNT100;
   1:  PR[GP1:91,1] = PR[GP1:90,1] + 27.157;
   1:  PR[GP1:91,2] = PR[GP1:90,2] + 17.534;
   1:L PR[91] R[100]mm/sec CNT100;
   1:  PR[GP1:91,1] = PR[GP1:90,1] + 24.231;
   1:  PR[GP1:91,2] = PR[GP1:90,2] + 18.592;
   1:L PR[91] R[100]mm/sec CNT100;
   1:  PR[GP1:91,1] = PR[GP1:90,1] + 20.982;
   1:  PR[GP1:91,2] = PR[GP1:90,2] + 19.264;
   1:L PR[91] R[100]mm/sec CNT100;
   1:  PR[GP1:91,1] = PR[GP1:90,1] + 20.758;
   1:  PR[GP1:91,2] = PR[GP1:90,2] + 19.290;
   1:L PR[91] R[100]mm/sec CNT100;
   1:  PR[GP1:91,1] = PR[GP1:90,1] + 17.520;
   1:  PR[GP1:91,2] = PR[GP1:90,2] + 19.459;
   1:L PR[91] R[100]mm/sec CNT100;
   1:  PR[GP1:91,1] = PR[GP1:90,1] + 14.634;
   1:  PR[GP1:91,2] = PR[GP1:90,2] + 19.166;
   1:L PR[91] R[100]mm/sec CNT100;
   1:  PR[GP1:91,1] = PR[GP1:90,1] + 13.768;
   1:  PR[GP1:91,2] = PR[GP1:90,2] + 19.046;
   1:L PR[91] R[100]mm/sec CNT100;
   1:  PR[GP1:91,1] = PR[GP1:90,1] + 11.095;
   1:  PR[GP1:91,2] = PR[GP1:90,2] + 18.353;
   1:L PR[91] R[100]mm/sec CNT100;
   1:  PR[GP1:91,1] = PR[GP1:90,1] + 8.749;
   1:  PR[GP1:91,2] = PR[GP1:90,2] + 17.327;
   1:L PR[91] R[100]mm/sec CNT100;
   1:  PR[GP1:91,1] = PR[GP1:90,1] + 7.438;
   1:  PR[GP1:91,2] = PR[GP1:90,2] + 16.779;
   1:L PR[91] R[100]mm/sec CNT100;
   1:  PR[GP1:91,1] = PR[GP1:90,1] + 5.424;
   1:  PR[GP1:91,2] = PR[GP1:90,2] + 15.493;
   1:L PR[91] R[100]mm/sec CNT100;
   1:  PR[GP1:91,1] = PR[GP1:90,1] + 5.171;
   1:  PR[GP1:91,2] = PR[GP1:90,2] + 15.318;
   1:L PR[91] R[100]mm/sec CNT100;
   1:  PR[GP1:91,1] = PR[GP1:90,1] + 4.692;
   1:  PR[GP1:91,2] = PR[GP1:90,2] + 14.939;
   1:L PR[91] R[100]mm/sec CNT100;
   1:  PR[GP1:91,1] = PR[GP1:90,1] + 3.034;
   1:  PR[GP1:91,2] = PR[GP1:90,2] + 13.458;
   1:L PR[91] R[100]mm/sec CNT100;
   1:  PR[GP1:91,1] = PR[GP1:90,1] + 2.330;
   1:  PR[GP1:91,2] = PR[GP1:90,2] + 12.730;
   1:L PR[91] R[100]mm/sec CNT100;
   1:  PR[GP1:91,1] = PR[GP1:90,1] + 2.090;
   1:  PR[GP1:91,2] = PR[GP1:90,2] + 12.413;
   1:L PR[91] R[100]mm/sec CNT100;
   1:  PR[GP1:91,1] = PR[GP1:90,1] + 1.443;
   1:  PR[GP1:91,2] = PR[GP1:90,2] + 11.955;
   1:L PR[91] R[100]mm/sec CNT100;
   1:  PR[GP1:91,1] = PR[GP1:90,1] + 0.740;
   1:  PR[GP1:91,2] = PR[GP1:90,2] + 11.570;
   1:L PR[91] R[100]mm/sec CNT100;
   1:  PR[GP1:91,1] = PR[GP1:90,1] + -0.586;
   1:L PR[91] R[100]mm/sec CNT100;
   1:  PR[91] = PR[90];
   1:  PR[GP1:91,1] = PR[GP1:90,1] + -1.541;
   1:  PR[GP1:91,2] = PR[GP1:90,2] + 12.321;
   1:  PR[GP1:91,3] = PR[GP1:90,3] + 28.365;
   1:L PR[91] R[100]mm/sec CNT100;
   1:  PR[GP1:91,1] = PR[GP1:90,1] + -1.870;
   1:  PR[GP1:91,2] = PR[GP1:90,2] + 12.749;
   1:L PR[91] R[100]mm/sec CNT100;
   1:  PR[GP1:91,1] = PR[GP1:90,1] + -2.109;
   1:  PR[GP1:91,2] = PR[GP1:90,2] + 12.974;
   1:L PR[91] R[100]mm/sec CNT100;
   1:  PR[GP1:91,1] = PR[GP1:90,1] + -2.678;
   1:  PR[GP1:91,2] = PR[GP1:90,2] + 13.569;
   1:L PR[91] R[100]mm/sec CNT100;
   1:  PR[GP1:91,1] = PR[GP1:90,1] + -4.236;
   1:  PR[GP1:91,2] = PR[GP1:90,2] + 14.958;
   1:L PR[91] R[100]mm/sec CNT100;
   1:  PR[GP1:91,1] = PR[GP1:90,1] + -4.761;
   1:  PR[GP1:91,2] = PR[GP1:90,2] + 15.373;
   1:L PR[91] R[100]mm/sec CNT100;
   1:  PR[GP1:91,1] = PR[GP1:90,1] + -6.588;
   1:  PR[GP1:91,2] = PR[GP1:90,2] + 16.543;
   1:L PR[91] R[100]mm/sec CNT100;
   1:  PR[GP1:91,1] = PR[GP1:90,1] + -7.022;
   1:  PR[GP1:91,2] = PR[GP1:90,2] + 16.834;
   1:L PR[91] R[100]mm/sec CNT100;
   1:  PR[GP1:91,1] = PR[GP1:90,1] + -9.377;
   1:  PR[GP1:91,2] = PR[GP1:90,2] + 17.863;
   1:L PR[91] R[100]mm/sec CNT100;
   1:  PR[GP1:91,1] = PR[GP1:90,1] + -10.739;
   1:  PR[GP1:91,2] = PR[GP1:90,2] + 18.434;
   1:L PR[91] R[100]mm/sec CNT100;
   1:  PR[GP1:91,1] = PR[GP1:90,1] + -13.266;
   1:  PR[GP1:91,2] = PR[GP1:90,2] + 19.087;
   1:L PR[91] R[100]mm/sec CNT100;
   1:  PR[GP1:91,1] = PR[GP1:90,1] + -16.330;
   1:  PR[GP1:91,2] = PR[GP1:90,2] + 19.406;
   1:L PR[91] R[100]mm/sec CNT100;
   1:  PR[GP1:91,1] = PR[GP1:90,1] + -17.174;
   1:  PR[GP1:91,2] = PR[GP1:90,2] + 19.521;
   1:L PR[91] R[100]mm/sec CNT100;
   1:  PR[GP1:91,1] = PR[GP1:90,1] + -20.260;
   1:  PR[GP1:91,2] = PR[GP1:90,2] + 19.358;
   1:L PR[91] R[100]mm/sec CNT100;
   1:  PR[GP1:91,1] = PR[GP1:90,1] + -20.724;
   1:  PR[GP1:91,2] = PR[GP1:90,2] + 19.304;
   1:L PR[91] R[100]mm/sec CNT100;
   1:  PR[GP1:91,1] = PR[GP1:90,1] + -23.832;
   1:  PR[GP1:91,2] = PR[GP1:90,2] + 18.659;
   1:L PR[91] R[100]mm/sec CNT100;
   1:  PR[GP1:91,1] = PR[GP1:90,1] + -26.964;
   1:  PR[GP1:91,2] = PR[GP1:90,2] + 17.504;
   1:L PR[91] R[100]mm/sec CNT100;
   1:  PR[GP1:91,1] = PR[GP1:90,1] + -29.926;
   1:  PR[GP1:91,2] = PR[GP1:90,2] + 15.872;
   1:L PR[91] R[100]mm/sec CNT100;
   1:  PR[GP1:91,1] = PR[GP1:90,1] + -30.643;
   1:  PR[GP1:91,2] = PR[GP1:90,2] + 15.268;
   1:L PR[91] R[100]mm/sec CNT100;
   1:  PR[GP1:91,1] = PR[GP1:90,1] + -32.892;
   1:  PR[GP1:91,2] = PR[GP1:90,2] + 13.488;
   1:L PR[91] R[100]mm/sec CNT100;
   1:  PR[GP1:91,1] = PR[GP1:90,1] + -34.331;
   1:  PR[GP1:91,2] = PR[GP1:90,2] + 11.939;
   1:L PR[91] R[100]mm/sec CNT100;
   1:  PR[GP1:91,1] = PR[GP1:90,1] + -35.417;
   1:  PR[GP1:91,2] = PR[GP1:90,2] + 10.423;
   1:L PR[91] R[100]mm/sec CNT100;
   1:  PR[GP1:91,1] = PR[GP1:90,1] + -36.499;
   1:  PR[GP1:91,2] = PR[GP1:90,2] + 8.777;
   1:L PR[91] R[100]mm/sec CNT100;
   1:  PR[GP1:91,1] = PR[GP1:90,1] + -37.206;
   1:  PR[GP1:91,2] = PR[GP1:90,2] + 7.190;
   1:L PR[91] R[100]mm/sec CNT100;
   1:  PR[GP1:91,1] = PR[GP1:90,1] + -38.062;
   1:  PR[GP1:91,2] = PR[GP1:90,2] + 5.058;
   1:L PR[91] R[100]mm/sec CNT100;
   1:  PR[GP1:91,1] = PR[GP1:90,1] + -38.428;
   1:  PR[GP1:91,2] = PR[GP1:90,2] + 3.643;
   1:L PR[91] R[100]mm/sec CNT100;
   1:  PR[GP1:91,1] = PR[GP1:90,1] + -38.751;
   1:  PR[GP1:91,2] = PR[GP1:90,2] + 1.099;
   1:L PR[91] R[100]mm/sec CNT100;
   1:  PR[GP1:91,1] = PR[GP1:90,1] + -38.860;
   1:  PR[GP1:91,2] = PR[GP1:90,2] + -0.277;
   1:L PR[91] R[100]mm/sec CNT100;
   1:  PR[GP1:91,1] = PR[GP1:90,1] + -38.538;
   1:  PR[GP1:91,2] = PR[GP1:90,2] + -2.788;
   1:L PR[91] R[100]mm/sec CNT100;
   1:  PR[GP1:91,1] = PR[GP1:90,1] + -38.420;
   1:  PR[GP1:91,2] = PR[GP1:90,2] + -4.301;
   1:L PR[91] R[100]mm/sec CNT100;
   1:  PR[GP1:91,1] = PR[GP1:90,1] + -38.062;
   1:  PR[GP1:91,2] = PR[GP1:90,2] + -5.682;
   1:L PR[91] R[100]mm/sec CNT100;
   1:  PR[GP1:91,1] = PR[GP1:90,1] + -37.206;
   1:  PR[GP1:91,2] = PR[GP1:90,2] + -7.814;
   1:L PR[91] R[100]mm/sec CNT100;
   1:  PR[GP1:91,1] = PR[GP1:90,1] + -36.512;
   1:  PR[GP1:91,2] = PR[GP1:90,2] + -9.372;
   1:L PR[91] R[100]mm/sec CNT100;
   1:  PR[GP1:91,1] = PR[GP1:90,1] + -35.356;
   1:  PR[GP1:91,2] = PR[GP1:90,2] + -10.976;
   1:L PR[91] R[100]mm/sec CNT100;
   1:  PR[GP1:91,1] = PR[GP1:90,1] + -34.309;
   1:  PR[GP1:91,2] = PR[GP1:90,2] + -12.587;
   1:L PR[91] R[100]mm/sec CNT100;
   1:  PR[GP1:91,1] = PR[GP1:90,1] + -32.875;
   1:  PR[GP1:91,2] = PR[GP1:90,2] + -14.130;
   1:L PR[91] R[100]mm/sec CNT100;
   1:  PR[GP1:91,1] = PR[GP1:90,1] + -31.875;
   1:  PR[GP1:91,2] = PR[GP1:90,2] + -14.979;
   1:L PR[91] R[100]mm/sec CNT100;
   1:  PR[GP1:91,1] = PR[GP1:90,1] + -29.950;
   1:  PR[GP1:91,2] = PR[GP1:90,2] + -16.483;
   1:L PR[91] R[100]mm/sec CNT100;
   1:  PR[GP1:91,1] = PR[GP1:90,1] + -26.964;
   1:  PR[GP1:91,2] = PR[GP1:90,2] + -18.128;
   1:L PR[91] R[100]mm/sec CNT100;
   1:  PR[GP1:91,1] = PR[GP1:90,1] + -23.830;
   1:  PR[GP1:91,2] = PR[GP1:90,2] + -19.283;
   1:L PR[91] R[100]mm/sec CNT100;
   1:  PR[GP1:91,1] = PR[GP1:90,1] + -20.722;
   1:  PR[GP1:91,2] = PR[GP1:90,2] + -19.928;
   1:L PR[91] R[100]mm/sec CNT100;
   1:  PR[GP1:91,1] = PR[GP1:90,1] + -20.256;
   1:  PR[GP1:91,2] = PR[GP1:90,2] + -19.982;
   1:L PR[91] R[100]mm/sec CNT100;
   1:  PR[GP1:91,1] = PR[GP1:90,1] + -17.142;
   1:  PR[GP1:91,2] = PR[GP1:90,2] + -20.146;
   1:L PR[91] R[100]mm/sec CNT100;
   1:  PR[GP1:91,1] = PR[GP1:90,1] + -14.376;
   1:  PR[GP1:91,2] = PR[GP1:90,2] + -19.868;
   1:L PR[91] R[100]mm/sec CNT100;
   1:  PR[GP1:91,1] = PR[GP1:90,1] + -13.279;
   1:  PR[GP1:91,2] = PR[GP1:90,2] + -19.714;
   1:L PR[91] R[100]mm/sec CNT100;
   1:  PR[GP1:91,1] = PR[GP1:90,1] + -10.738;
   1:  PR[GP1:91,2] = PR[GP1:90,2] + -19.057;
   1:L PR[91] R[100]mm/sec CNT100;
   1:  PR[GP1:91,1] = PR[GP1:90,1] + -8.500;
   1:  PR[GP1:91,2] = PR[GP1:90,2] + -18.076;
   1:L PR[91] R[100]mm/sec CNT100;
   1:  PR[GP1:91,1] = PR[GP1:90,1] + -6.954;
   1:  PR[GP1:91,2] = PR[GP1:90,2] + -17.417;
   1:L PR[91] R[100]mm/sec CNT100;
   1:  PR[GP1:91,1] = PR[GP1:90,1] + -5.052;
   1:  PR[GP1:91,2] = PR[GP1:90,2] + -16.201;
   1:L PR[91] R[100]mm/sec CNT100;
   1:  PR[GP1:91,1] = PR[GP1:90,1] + -4.596;
   1:  PR[GP1:91,2] = PR[GP1:90,2] + -15.871;
   1:L PR[91] R[100]mm/sec CNT100;
   1:  PR[GP1:91,1] = PR[GP1:90,1] + -2.999;
   1:  PR[GP1:91,2] = PR[GP1:90,2] + -14.474;
   1:L PR[91] R[100]mm/sec CNT100;
   1:  PR[GP1:91,1] = PR[GP1:90,1] + -2.567;
   1:  PR[GP1:91,2] = PR[GP1:90,2] + -14.085;
   1:L PR[91] R[100]mm/sec CNT100;
   1:  PR[GP1:91,1] = PR[GP1:90,1] + -2.101;
   1:  PR[GP1:91,2] = PR[GP1:90,2] + -13.539;
   1:L PR[91] R[100]mm/sec CNT100;
   1:  PR[GP1:91,1] = PR[GP1:90,1] + -1.599;
   1:  PR[GP1:91,2] = PR[GP1:90,2] + -13.135;
   1:L PR[91] R[100]mm/sec CNT100;
   1:  PR[GP1:91,1] = PR[GP1:90,1] + -0.477;
   1:  PR[GP1:91,2] = PR[GP1:90,2] + -12.341;
   1:L PR[91] R[100]mm/sec CNT100;
   1:  PR[GP1:91,1] = PR[GP1:90,1] + 0.564;
   1:  PR[GP1:91,2] = PR[GP1:90,2] + -12.711;
   1:L PR[91] R[100]mm/sec CNT100;
   1:  PR[GP1:91,1] = PR[GP1:90,1] + 1.217;
   1:L PR[91] R[100]mm/sec CNT100;
   1:  PR[GP1:91,1] = PR[GP1:90,1] + 1.898;
   1:  PR[GP1:91,2] = PR[GP1:90,2] + -13.268;
   1:L PR[91] R[100]mm/sec CNT100;
   1:  PR[GP1:91,1] = PR[GP1:90,1] + 2.236;
   1:  PR[GP1:91,2] = PR[GP1:90,2] + -13.509;
   1:L PR[91] R[100]mm/sec CNT100;
   1:  PR[GP1:91,1] = PR[GP1:90,1] + 2.727;
   1:  PR[GP1:91,2] = PR[GP1:90,2] + -14.086;
   1:L PR[91] R[100]mm/sec CNT100;
   1:  PR[GP1:91,1] = PR[GP1:90,1] + 4.736;
   1:  PR[GP1:91,2] = PR[GP1:90,2] + -15.859;
   1:L PR[91] R[100]mm/sec CNT100;
   1:  PR[GP1:91,1] = PR[GP1:90,1] + 6.403;
   1:  PR[GP1:91,2] = PR[GP1:90,2] + -16.926;
   1:L PR[91] R[100]mm/sec CNT100;
   1:  PR[GP1:91,1] = PR[GP1:90,1] + 7.134;
   1:  PR[GP1:91,2] = PR[GP1:90,2] + -17.430;
   1:L PR[91] R[100]mm/sec CNT100;
   1:  PR[GP1:91,1] = PR[GP1:90,1] + 10.884;
   1:  PR[GP1:91,2] = PR[GP1:90,2] + -19.052;
   1:L PR[91] R[100]mm/sec CNT100;
   1:  PR[GP1:91,1] = PR[GP1:90,1] + 13.409;
   1:  PR[GP1:91,2] = PR[GP1:90,2] + -19.707;
   1:L PR[91] R[100]mm/sec CNT100;
   1:  PR[GP1:91,1] = PR[GP1:90,1] + 16.470;
   1:  PR[GP1:91,2] = PR[GP1:90,2] + -20.028;
   1:L PR[91] R[100]mm/sec CNT100;
   1:  PR[GP1:91,1] = PR[GP1:90,1] + 17.317;
   1:  PR[GP1:91,2] = PR[GP1:90,2] + -20.145;
   1:L PR[91] R[100]mm/sec CNT100;
   1:  PR[GP1:91,1] = PR[GP1:90,1] + 20.388;
   1:  PR[GP1:91,2] = PR[GP1:90,2] + -19.986;
   1:L PR[91] R[100]mm/sec CNT100;
   1:  PR[GP1:91,1] = PR[GP1:90,1] + 20.856;
   1:  PR[GP1:91,2] = PR[GP1:90,2] + -19.931;
   1:L PR[91] R[100]mm/sec CNT100;
   1:  PR[GP1:91,1] = PR[GP1:90,1] + 23.960;
   1:  PR[GP1:91,2] = PR[GP1:90,2] + -19.289;
   1:L PR[91] R[100]mm/sec CNT100;
   1:  PR[GP1:91,1] = PR[GP1:90,1] + 27.104;
   1:  PR[GP1:91,2] = PR[GP1:90,2] + -18.135;
   1:L PR[91] R[100]mm/sec CNT100;
   1:  PR[GP1:91,1] = PR[GP1:90,1] + 30.057;
   1:  PR[GP1:91,2] = PR[GP1:90,2] + -16.516;
   1:L PR[91] R[100]mm/sec CNT100;
   1:  PR[GP1:91,1] = PR[GP1:90,1] + 30.770;
   1:  PR[GP1:91,2] = PR[GP1:90,2] + -15.915;
   1:L PR[91] R[100]mm/sec CNT100;
   1:  PR[GP1:91,1] = PR[GP1:90,1] + 33.013;
   1:  PR[GP1:91,2] = PR[GP1:90,2] + -14.145;
   1:L PR[91] R[100]mm/sec CNT100;
   1:  PR[GP1:91,1] = PR[GP1:90,1] + 34.463;
   1:  PR[GP1:91,2] = PR[GP1:90,2] + -12.587;
   1:L PR[91] R[100]mm/sec CNT100;
   1:  PR[GP1:91,1] = PR[GP1:90,1] + 35.549;
   1:  PR[GP1:91,2] = PR[GP1:90,2] + -11.071;
   1:L PR[91] R[100]mm/sec CNT100;
   1:  PR[GP1:91,1] = PR[GP1:90,1] + 36.650;
   1:  PR[GP1:91,2] = PR[GP1:90,2] + -9.405;
   1:L PR[91] R[100]mm/sec CNT100;
   1:  PR[GP1:91,1] = PR[GP1:90,1] + 37.356;
   1:  PR[GP1:91,2] = PR[GP1:90,2] + -7.841;
   1:L PR[91] R[100]mm/sec CNT100;
   1:  PR[GP1:91,1] = PR[GP1:90,1] + 38.211;
   1:  PR[GP1:91,2] = PR[GP1:90,2] + -5.722;
   1:L PR[91] R[100]mm/sec CNT100;
   1:  PR[GP1:91,1] = PR[GP1:90,1] + 38.578;
   1:  PR[GP1:91,2] = PR[GP1:90,2] + -4.323;
   1:L PR[91] R[100]mm/sec CNT100;
   1:  PR[GP1:91,1] = PR[GP1:90,1] + 38.901;
   1:  PR[GP1:91,2] = PR[GP1:90,2] + -1.769;
   1:L PR[91] R[100]mm/sec CNT100;
   1:  PR[GP1:91,1] = PR[GP1:90,1] + 39.016;
   1:  PR[GP1:91,2] = PR[GP1:90,2] + -0.345;
   1:L PR[91] R[100]mm/sec CNT100;
   1:  PR[GP1:91,1] = PR[GP1:90,1] + 38.695;
   1:  PR[GP1:91,2] = PR[GP1:90,2] + 2.173;
   1:L PR[91] R[100]mm/sec CNT100;
   1:  PR[GP1:91,1] = PR[GP1:90,1] + 38.570;
   1:  PR[GP1:91,2] = PR[GP1:90,2] + 3.732;
   1:L PR[91] R[100]mm/sec CNT100;
   1:  PR[GP1:91,1] = PR[GP1:90,1] + 38.211;
   1:  PR[GP1:91,2] = PR[GP1:90,2] + 5.098;
   1:L PR[91] R[100]mm/sec CNT100;
   1:  PR[GP1:91,1] = PR[GP1:90,1] + 37.355;
   1:  PR[GP1:91,2] = PR[GP1:90,2] + 7.219;
   1:L PR[91] R[100]mm/sec CNT100;
   1:  PR[GP1:91,1] = PR[GP1:90,1] + 36.661;
   1:  PR[GP1:91,2] = PR[GP1:90,2] + 8.756;
   1:L PR[91] R[100]mm/sec CNT100;
   1:  PR[GP1:91,1] = PR[GP1:90,1] + 35.505;
   1:  PR[GP1:91,2] = PR[GP1:90,2] + 10.362;
   1:L PR[91] R[100]mm/sec CNT100;
   1:  PR[GP1:91,1] = PR[GP1:90,1] + 34.441;
   1:  PR[GP1:91,2] = PR[GP1:90,2] + 11.987;
   1:L PR[91] R[100]mm/sec CNT100;
   1:  PR[GP1:91,1] = PR[GP1:90,1] + 32.994;
   1:  PR[GP1:91,2] = PR[GP1:90,2] + 13.541;
   1:L PR[91] R[100]mm/sec CNT100;
   1:  PR[GP1:91,1] = PR[GP1:90,1] + 31.998;
   1:  PR[GP1:91,2] = PR[GP1:90,2] + 14.388;
   1:L PR[91] R[100]mm/sec CNT100;
   1:  PR[GP1:91,1] = PR[GP1:90,1] + 30.082;
   1:  PR[GP1:91,2] = PR[GP1:90,2] + 15.879;
   1:L PR[91] R[100]mm/sec CNT100;
   1:  PR[GP1:91,1] = PR[GP1:90,1] + 27.103;
   1:  PR[GP1:91,2] = PR[GP1:90,2] + 17.511;
   1:L PR[91] R[100]mm/sec CNT100;
   1:  PR[GP1:91,1] = PR[GP1:90,1] + 23.962;
   1:  PR[GP1:91,2] = PR[GP1:90,2] + 18.664;
   1:L PR[91] R[100]mm/sec CNT100;
   1:  PR[GP1:91,1] = PR[GP1:90,1] + 20.858;
   1:  PR[GP1:91,2] = PR[GP1:90,2] + 19.307;
   1:L PR[91] R[100]mm/sec CNT100;
   1:  PR[GP1:91,1] = PR[GP1:90,1] + 20.392;
   1:  PR[GP1:91,2] = PR[GP1:90,2] + 19.362;
   1:L PR[91] R[100]mm/sec CNT100;
   1:  PR[GP1:91,1] = PR[GP1:90,1] + 17.296;
   1:  PR[GP1:91,2] = PR[GP1:90,2] + 19.523;
   1:L PR[91] R[100]mm/sec CNT100;
   1:  PR[GP1:91,1] = PR[GP1:90,1] + 14.537;
   1:  PR[GP1:91,2] = PR[GP1:90,2] + 19.243;
   1:L PR[91] R[100]mm/sec CNT100;
   1:  PR[GP1:91,1] = PR[GP1:90,1] + 13.443;
   1:  PR[GP1:91,2] = PR[GP1:90,2] + 19.092;
   1:L PR[91] R[100]mm/sec CNT100;
   1:  PR[GP1:91,1] = PR[GP1:90,1] + 10.900;
   1:  PR[GP1:91,2] = PR[GP1:90,2] + 18.432;
   1:L PR[91] R[100]mm/sec CNT100;
   1:  PR[GP1:91,1] = PR[GP1:90,1] + 8.663;
   1:  PR[GP1:91,2] = PR[GP1:90,2] + 17.454;
   1:L PR[91] R[100]mm/sec CNT100;
   1:  PR[GP1:91,1] = PR[GP1:90,1] + 7.150;
   1:  PR[GP1:91,2] = PR[GP1:90,2] + 16.822;
   1:L PR[91] R[100]mm/sec CNT100;
   1:  PR[GP1:91,1] = PR[GP1:90,1] + 5.242;
   1:  PR[GP1:91,2] = PR[GP1:90,2] + 15.603;
   1:L PR[91] R[100]mm/sec CNT100;
   1:  PR[GP1:91,1] = PR[GP1:90,1] + 4.950;
   1:  PR[GP1:91,2] = PR[GP1:90,2] + 15.401;
   1:L PR[91] R[100]mm/sec CNT100;
   1:  PR[GP1:91,1] = PR[GP1:90,1] + 4.403;
   1:  PR[GP1:91,2] = PR[GP1:90,2] + 14.969;
   1:L PR[91] R[100]mm/sec CNT100;
   1:  PR[GP1:91,1] = PR[GP1:90,1] + 2.844;
   1:  PR[GP1:91,2] = PR[GP1:90,2] + 13.578;
   1:L PR[91] R[100]mm/sec CNT100;
   1:  PR[GP1:91,1] = PR[GP1:90,1] + 2.206;
   1:  PR[GP1:91,2] = PR[GP1:90,2] + 12.907;
   1:L PR[91] R[100]mm/sec CNT100;
   1:  PR[GP1:91,1] = PR[GP1:90,1] + 2.161;
   1:  PR[GP1:91,2] = PR[GP1:90,2] + 12.875;
   1:L PR[91] R[100]mm/sec CNT100;
   1:  PR[GP1:91,1] = PR[GP1:90,1] + 2.032;
   1:  PR[GP1:91,2] = PR[GP1:90,2] + 12.705;
   1:L PR[91] R[100]mm/sec CNT100;
   1:  PR[GP1:91,1] = PR[GP1:90,1] + 1.467;
   1:  PR[GP1:91,2] = PR[GP1:90,2] + 12.305;
   1:L PR[91] R[100]mm/sec CNT100;
   1:  PR[GP1:91,1] = PR[GP1:90,1] + 0.699;
   1:  PR[GP1:91,2] = PR[GP1:90,2] + 11.885;
   1:L PR[91] R[100]mm/sec CNT100;
   1:  PR[GP1:91,1] = PR[GP1:90,1] + -0.562;
   1:  PR[GP1:91,2] = PR[GP1:90,2] + 11.884;
   1:L PR[91] R[100]mm/sec CNT100;
   1:  PR[91] = PR[90];
   1:  PR[GP1:91,1] = PR[GP1:90,1] + -1.580;
   1:  PR[GP1:91,2] = PR[GP1:90,2] + 12.664;
   1:  PR[GP1:91,3] = PR[GP1:90,3] + 28.975;
   1:L PR[91] R[100]mm/sec CNT100;
   1:  PR[GP1:91,1] = PR[GP1:90,1] + -1.940;
   1:  PR[GP1:91,2] = PR[GP1:90,2] + 13.132;
   1:L PR[91] R[100]mm/sec CNT100;
   1:  PR[GP1:91,1] = PR[GP1:90,1] + -2.091;
   1:  PR[GP1:91,2] = PR[GP1:90,2] + 13.274;
   1:L PR[91] R[100]mm/sec CNT100;
   1:  PR[GP1:91,1] = PR[GP1:90,1] + -2.485;
   1:  PR[GP1:91,2] = PR[GP1:90,2] + 13.687;
   1:L PR[91] R[100]mm/sec CNT100;
   1:  PR[GP1:91,1] = PR[GP1:90,1] + -3.950;
   1:  PR[GP1:91,2] = PR[GP1:90,2] + 14.989;
   1:L PR[91] R[100]mm/sec CNT100;
   1:  PR[GP1:91,1] = PR[GP1:90,1] + -4.541;
   1:  PR[GP1:91,2] = PR[GP1:90,2] + 15.457;
   1:L PR[91] R[100]mm/sec CNT100;
   1:  PR[GP1:91,1] = PR[GP1:90,1] + -6.235;
   1:  PR[GP1:91,2] = PR[GP1:90,2] + 16.541;
   1:L PR[91] R[100]mm/sec CNT100;
   1:  PR[GP1:91,1] = PR[GP1:90,1] + -6.735;
   1:  PR[GP1:91,2] = PR[GP1:90,2] + 16.877;
   1:L PR[91] R[100]mm/sec CNT100;
   1:  PR[GP1:91,1] = PR[GP1:90,1] + -8.963;
   1:  PR[GP1:91,2] = PR[GP1:90,2] + 17.850;
   1:L PR[91] R[100]mm/sec CNT100;
   1:  PR[GP1:91,1] = PR[GP1:90,1] + -10.543;
   1:  PR[GP1:91,2] = PR[GP1:90,2] + 18.513;
   1:L PR[91] R[100]mm/sec CNT100;
   1:  PR[GP1:91,1] = PR[GP1:90,1] + -12.941;
   1:  PR[GP1:91,2] = PR[GP1:90,2] + 19.133;
   1:L PR[91] R[100]mm/sec CNT100;
   1:  PR[GP1:91,1] = PR[GP1:90,1] + -15.857;
   1:  PR[GP1:91,2] = PR[GP1:90,2] + 19.436;
   1:L PR[91] R[100]mm/sec CNT100;
   1:  PR[GP1:91,1] = PR[GP1:90,1] + -16.950;
   1:  PR[GP1:91,2] = PR[GP1:90,2] + 19.585;
   1:L PR[91] R[100]mm/sec CNT100;
   1:  PR[GP1:91,1] = PR[GP1:90,1] + -19.892;
   1:  PR[GP1:91,2] = PR[GP1:90,2] + 19.430;
   1:L PR[91] R[100]mm/sec CNT100;
   1:  PR[GP1:91,1] = PR[GP1:90,1] + -20.599;
   1:  PR[GP1:91,2] = PR[GP1:90,2] + 19.346;
   1:L PR[91] R[100]mm/sec CNT100;
   1:  PR[GP1:91,1] = PR[GP1:90,1] + -23.571;
   1:  PR[GP1:91,2] = PR[GP1:90,2] + 18.730;
   1:L PR[91] R[100]mm/sec CNT100;
   1:  PR[GP1:91,1] = PR[GP1:90,1] + -26.859;
   1:  PR[GP1:91,2] = PR[GP1:90,2] + 17.507;
   1:L PR[91] R[100]mm/sec CNT100;
   1:  PR[GP1:91,1] = PR[GP1:90,1] + -29.739;
   1:  PR[GP1:91,2] = PR[GP1:90,2] + 15.903;
   1:L PR[91] R[100]mm/sec CNT100;
   1:  PR[GP1:91,1] = PR[GP1:90,1] + -29.993;
   1:  PR[GP1:91,2] = PR[GP1:90,2] + 15.689;
   1:L PR[91] R[100]mm/sec CNT100;
   1:  PR[GP1:91,1] = PR[GP1:90,1] + -32.584;
   1:  PR[GP1:91,2] = PR[GP1:90,2] + 13.638;
   1:L PR[91] R[100]mm/sec CNT100;
   1:  PR[GP1:91,1] = PR[GP1:90,1] + -34.255;
   1:  PR[GP1:91,2] = PR[GP1:90,2] + 11.840;
   1:L PR[91] R[100]mm/sec CNT100;
   1:  PR[GP1:91,1] = PR[GP1:90,1] + -35.041;
   1:  PR[GP1:91,2] = PR[GP1:90,2] + 10.743;
   1:L PR[91] R[100]mm/sec CNT100;
   1:  PR[GP1:91,1] = PR[GP1:90,1] + -36.322;
   1:  PR[GP1:91,2] = PR[GP1:90,2] + 8.794;
   1:L PR[91] R[100]mm/sec CNT100;
   1:  PR[GP1:91,1] = PR[GP1:90,1] + -37.160;
   1:  PR[GP1:91,2] = PR[GP1:90,2] + 6.913;
   1:L PR[91] R[100]mm/sec CNT100;
   1:  PR[GP1:91,1] = PR[GP1:90,1] + -37.845;
   1:  PR[GP1:91,2] = PR[GP1:90,2] + 5.208;
   1:L PR[91] R[100]mm/sec CNT100;
   1:  PR[GP1:91,1] = PR[GP1:90,1] + -38.289;
   1:  PR[GP1:91,2] = PR[GP1:90,2] + 3.489;
   1:L PR[91] R[100]mm/sec CNT100;
   1:  PR[GP1:91,1] = PR[GP1:90,1] + -38.551;
   1:  PR[GP1:91,2] = PR[GP1:90,2] + 1.422;
   1:L PR[91] R[100]mm/sec CNT100;
   1:  PR[GP1:91,1] = PR[GP1:90,1] + -38.686;
   1:  PR[GP1:91,2] = PR[GP1:90,2] + -0.277;
   1:L PR[91] R[100]mm/sec CNT100;
   1:  PR[GP1:91,1] = PR[GP1:90,1] + -38.423;
   1:  PR[GP1:91,2] = PR[GP1:90,2] + -2.328;
   1:L PR[91] R[100]mm/sec CNT100;
   1:  PR[GP1:91,1] = PR[GP1:90,1] + -38.280;
   1:  PR[GP1:91,2] = PR[GP1:90,2] + -4.147;
   1:L PR[91] R[100]mm/sec CNT100;
   1:  PR[GP1:91,1] = PR[GP1:90,1] + -37.845;
   1:  PR[GP1:91,2] = PR[GP1:90,2] + -5.832;
   1:L PR[91] R[100]mm/sec CNT100;
   1:  PR[GP1:91,1] = PR[GP1:90,1] + -37.160;
   1:  PR[GP1:91,2] = PR[GP1:90,2] + -7.537;
   1:L PR[91] R[100]mm/sec CNT100;
   1:  PR[GP1:91,1] = PR[GP1:90,1] + -36.335;
   1:  PR[GP1:91,2] = PR[GP1:90,2] + -9.389;
   1:L PR[91] R[100]mm/sec CNT100;
   1:  PR[GP1:91,1] = PR[GP1:90,1] + -35.442;
   1:  PR[GP1:91,2] = PR[GP1:90,2] + -10.629;
   1:L PR[91] R[100]mm/sec CNT100;
   1:  PR[GP1:91,1] = PR[GP1:90,1] + -34.233;
   1:  PR[GP1:91,2] = PR[GP1:90,2] + -12.488;
   1:L PR[91] R[100]mm/sec CNT100;
   1:  PR[GP1:91,1] = PR[GP1:90,1] + -32.567;
   1:  PR[GP1:91,2] = PR[GP1:90,2] + -14.280;
   1:L PR[91] R[100]mm/sec CNT100;
   1:  PR[GP1:91,1] = PR[GP1:90,1] + -31.944;
   1:  PR[GP1:91,2] = PR[GP1:90,2] + -14.809;
   1:L PR[91] R[100]mm/sec CNT100;
   1:  PR[GP1:91,1] = PR[GP1:90,1] + -29.763;
   1:  PR[GP1:91,2] = PR[GP1:90,2] + -16.514;
   1:L PR[91] R[100]mm/sec CNT100;
   1:  PR[GP1:91,1] = PR[GP1:90,1] + -26.858;
   1:  PR[GP1:91,2] = PR[GP1:90,2] + -18.131;
   1:L PR[91] R[100]mm/sec CNT100;
   1:  PR[GP1:91,1] = PR[GP1:90,1] + -23.568;
   1:  PR[GP1:91,2] = PR[GP1:90,2] + -19.354;
   1:L PR[91] R[100]mm/sec CNT100;
   1:  PR[GP1:91,1] = PR[GP1:90,1] + -20.595;
   1:  PR[GP1:91,2] = PR[GP1:90,2] + -19.971;
   1:L PR[91] R[100]mm/sec CNT100;
   1:  PR[GP1:91,1] = PR[GP1:90,1] + -19.887;
   1:  PR[GP1:91,2] = PR[GP1:90,2] + -20.054;
   1:L PR[91] R[100]mm/sec CNT100;
   1:  PR[GP1:91,1] = PR[GP1:90,1] + -16.916;
   1:  PR[GP1:91,2] = PR[GP1:90,2] + -20.211;
   1:L PR[91] R[100]mm/sec CNT100;
   1:  PR[GP1:91,1] = PR[GP1:90,1] + -14.277;
   1:  PR[GP1:91,2] = PR[GP1:90,2] + -19.945;
   1:L PR[91] R[100]mm/sec CNT100;
   1:  PR[GP1:91,1] = PR[GP1:90,1] + -12.953;
   1:  PR[GP1:91,2] = PR[GP1:90,2] + -19.759;
   1:L PR[91] R[100]mm/sec CNT100;
   1:  PR[GP1:91,1] = PR[GP1:90,1] + -10.540;
   1:  PR[GP1:91,2] = PR[GP1:90,2] + -19.136;
   1:L PR[91] R[100]mm/sec CNT100;
   1:  PR[GP1:91,1] = PR[GP1:90,1] + -8.413;
   1:  PR[GP1:91,2] = PR[GP1:90,2] + -18.203;
   1:L PR[91] R[100]mm/sec CNT100;
   1:  PR[GP1:91,1] = PR[GP1:90,1] + -6.661;
   1:  PR[GP1:91,2] = PR[GP1:90,2] + -17.456;
   1:L PR[91] R[100]mm/sec CNT100;
   1:  PR[GP1:91,1] = PR[GP1:90,1] + -4.867;
   1:  PR[GP1:91,2] = PR[GP1:90,2] + -16.309;
   1:L PR[91] R[100]mm/sec CNT100;
   1:  PR[GP1:91,1] = PR[GP1:90,1] + -4.353;
   1:  PR[GP1:91,2] = PR[GP1:90,2] + -15.938;
   1:L PR[91] R[100]mm/sec CNT100;
   1:  PR[GP1:91,1] = PR[GP1:90,1] + -2.355;
   1:  PR[GP1:91,2] = PR[GP1:90,2] + -14.182;
   1:L PR[91] R[100]mm/sec CNT100;
   1:  PR[GP1:91,1] = PR[GP1:90,1] + -2.083;
   1:  PR[GP1:91,2] = PR[GP1:90,2] + -13.863;
   1:L PR[91] R[100]mm/sec CNT100;
   1:  PR[GP1:91,1] = PR[GP1:90,1] + -1.522;
   1:  PR[GP1:91,2] = PR[GP1:90,2] + -13.413;
   1:L PR[91] R[100]mm/sec CNT100;
   1:  PR[GP1:91,1] = PR[GP1:90,1] + -0.452;
   1:  PR[GP1:91,2] = PR[GP1:90,2] + -12.656;
   1:L PR[91] R[100]mm/sec CNT100;
   1:  PR[GP1:91,1] = PR[GP1:90,1] + 0.687;
   1:  PR[GP1:91,2] = PR[GP1:90,2] + -13.061;
   1:L PR[91] R[100]mm/sec CNT100;
   1:  PR[GP1:91,1] = PR[GP1:90,1] + 1.228;
   1:L PR[91] R[100]mm/sec CNT100;
   1:  PR[GP1:91,1] = PR[GP1:90,1] + 2.241;
   1:  PR[GP1:91,2] = PR[GP1:90,2] + -13.861;
   1:L PR[91] R[100]mm/sec CNT100;
   1:  PR[GP1:91,1] = PR[GP1:90,1] + 2.519;
   1:  PR[GP1:91,2] = PR[GP1:90,2] + -14.188;
   1:L PR[91] R[100]mm/sec CNT100;
   1:  PR[GP1:91,1] = PR[GP1:90,1] + 4.490;
   1:  PR[GP1:91,2] = PR[GP1:90,2] + -15.923;
   1:L PR[91] R[100]mm/sec CNT100;
   1:  PR[GP1:91,1] = PR[GP1:90,1] + 6.006;
   1:  PR[GP1:91,2] = PR[GP1:90,2] + -16.894;
   1:L PR[91] R[100]mm/sec CNT100;
   1:  PR[GP1:91,1] = PR[GP1:90,1] + 6.840;
   1:  PR[GP1:91,2] = PR[GP1:90,2] + -17.469;
   1:L PR[91] R[100]mm/sec CNT100;
   1:  PR[GP1:91,1] = PR[GP1:90,1] + 10.686;
   1:  PR[GP1:91,2] = PR[GP1:90,2] + -19.130;
   1:L PR[91] R[100]mm/sec CNT100;
   1:  PR[GP1:91,1] = PR[GP1:90,1] + 13.082;
   1:  PR[GP1:91,2] = PR[GP1:90,2] + -19.752;
   1:L PR[91] R[100]mm/sec CNT100;
   1:  PR[GP1:91,1] = PR[GP1:90,1] + 15.994;
   1:  PR[GP1:91,2] = PR[GP1:90,2] + -20.057;
   1:L PR[91] R[100]mm/sec CNT100;
   1:  PR[GP1:91,1] = PR[GP1:90,1] + 17.091;
   1:  PR[GP1:91,2] = PR[GP1:90,2] + -20.209;
   1:L PR[91] R[100]mm/sec CNT100;
   1:  PR[GP1:91,1] = PR[GP1:90,1] + 20.020;
   1:  PR[GP1:91,2] = PR[GP1:90,2] + -20.057;
   1:L PR[91] R[100]mm/sec CNT100;
   1:  PR[GP1:91,1] = PR[GP1:90,1] + 20.730;
   1:  PR[GP1:91,2] = PR[GP1:90,2] + -19.975;
   1:L PR[91] R[100]mm/sec CNT100;
   1:  PR[GP1:91,1] = PR[GP1:90,1] + 23.699;
   1:  PR[GP1:91,2] = PR[GP1:90,2] + -19.360;
   1:L PR[91] R[100]mm/sec CNT100;
   1:  PR[GP1:91,1] = PR[GP1:90,1] + 26.996;
   1:  PR[GP1:91,2] = PR[GP1:90,2] + -18.139;
   1:L PR[91] R[100]mm/sec CNT100;
   1:  PR[GP1:91,1] = PR[GP1:90,1] + 29.867;
   1:  PR[GP1:91,2] = PR[GP1:90,2] + -16.549;
   1:L PR[91] R[100]mm/sec CNT100;
   1:  PR[GP1:91,1] = PR[GP1:90,1] + 30.115;
   1:  PR[GP1:91,2] = PR[GP1:90,2] + -16.340;
   1:L PR[91] R[100]mm/sec CNT100;
   1:  PR[GP1:91,1] = PR[GP1:90,1] + 32.699;
   1:  PR[GP1:91,2] = PR[GP1:90,2] + -14.301;
   1:L PR[91] R[100]mm/sec CNT100;
   1:  PR[GP1:91,1] = PR[GP1:90,1] + 34.384;
   1:  PR[GP1:91,2] = PR[GP1:90,2] + -12.492;
   1:L PR[91] R[100]mm/sec CNT100;
   1:  PR[GP1:91,1] = PR[GP1:90,1] + 35.168;
   1:  PR[GP1:91,2] = PR[GP1:90,2] + -11.397;
   1:L PR[91] R[100]mm/sec CNT100;
   1:  PR[GP1:91,1] = PR[GP1:90,1] + 36.471;
   1:  PR[GP1:91,2] = PR[GP1:90,2] + -9.425;
   1:L PR[91] R[100]mm/sec CNT100;
   1:  PR[GP1:91,1] = PR[GP1:90,1] + 37.308;
   1:  PR[GP1:91,2] = PR[GP1:90,2] + -7.571;
   1:L PR[91] R[100]mm/sec CNT100;
   1:  PR[GP1:91,1] = PR[GP1:90,1] + 37.992;
   1:  PR[GP1:91,2] = PR[GP1:90,2] + -5.876;
   1:L PR[91] R[100]mm/sec CNT100;
   1:  PR[GP1:91,1] = PR[GP1:90,1] + 38.438;
   1:  PR[GP1:91,2] = PR[GP1:90,2] + -4.177;
   1:L PR[91] R[100]mm/sec CNT100;
   1:  PR[GP1:91,1] = PR[GP1:90,1] + 38.700;
   1:  PR[GP1:91,2] = PR[GP1:90,2] + -2.102;
   1:L PR[91] R[100]mm/sec CNT100;
   1:  PR[GP1:91,1] = PR[GP1:90,1] + 38.842;
   1:  PR[GP1:91,2] = PR[GP1:90,2] + -0.345;
   1:L PR[91] R[100]mm/sec CNT100;
   1:  PR[GP1:91,1] = PR[GP1:90,1] + 38.580;
   1:  PR[GP1:91,2] = PR[GP1:90,2] + 1.712;
   1:L PR[91] R[100]mm/sec CNT100;
   1:  PR[GP1:91,1] = PR[GP1:90,1] + 38.429;
   1:  PR[GP1:91,2] = PR[GP1:90,2] + 3.585;
   1:L PR[91] R[100]mm/sec CNT100;
   1:  PR[GP1:91,1] = PR[GP1:90,1] + 37.992;
   1:  PR[GP1:91,2] = PR[GP1:90,2] + 5.253;
   1:L PR[91] R[100]mm/sec CNT100;
   1:  PR[GP1:91,1] = PR[GP1:90,1] + 37.308;
   1:  PR[GP1:91,2] = PR[GP1:90,2] + 6.948;
   1:L PR[91] R[100]mm/sec CNT100;
   1:  PR[GP1:91,1] = PR[GP1:90,1] + 36.483;
   1:  PR[GP1:91,2] = PR[GP1:90,2] + 8.775;
   1:L PR[91] R[100]mm/sec CNT100;
   1:  PR[GP1:91,1] = PR[GP1:90,1] + 35.589;
   1:  PR[GP1:91,2] = PR[GP1:90,2] + 10.016;
   1:L PR[91] R[100]mm/sec CNT100;
   1:  PR[GP1:91,1] = PR[GP1:90,1] + 34.362;
   1:  PR[GP1:91,2] = PR[GP1:90,2] + 11.891;
   1:L PR[91] R[100]mm/sec CNT100;
   1:  PR[GP1:91,1] = PR[GP1:90,1] + 32.681;
   1:  PR[GP1:91,2] = PR[GP1:90,2] + 13.697;
   1:L PR[91] R[100]mm/sec CNT100;
   1:  PR[GP1:91,1] = PR[GP1:90,1] + 32.064;
   1:  PR[GP1:91,2] = PR[GP1:90,2] + 14.222;
   1:L PR[91] R[100]mm/sec CNT100;
   1:  PR[GP1:91,1] = PR[GP1:90,1] + 29.892;
   1:  PR[GP1:91,2] = PR[GP1:90,2] + 15.911;
   1:L PR[91] R[100]mm/sec CNT100;
   1:  PR[GP1:91,1] = PR[GP1:90,1] + 26.997;
   1:  PR[GP1:91,2] = PR[GP1:90,2] + 17.515;
   1:L PR[91] R[100]mm/sec CNT100;
   1:  PR[GP1:91,1] = PR[GP1:90,1] + 23.702;
   1:  PR[GP1:91,2] = PR[GP1:90,2] + 18.735;
   1:L PR[91] R[100]mm/sec CNT100;
   1:  PR[GP1:91,1] = PR[GP1:90,1] + 20.734;
   1:  PR[GP1:91,2] = PR[GP1:90,2] + 19.350;
   1:L PR[91] R[100]mm/sec CNT100;
   1:  PR[GP1:91,1] = PR[GP1:90,1] + 20.026;
   1:  PR[GP1:91,2] = PR[GP1:90,2] + 19.433;
   1:L PR[91] R[100]mm/sec CNT100;
   1:  PR[GP1:91,1] = PR[GP1:90,1] + 17.073;
   1:  PR[GP1:91,2] = PR[GP1:90,2] + 19.587;
   1:L PR[91] R[100]mm/sec CNT100;
   1:  PR[GP1:91,1] = PR[GP1:90,1] + 14.440;
   1:  PR[GP1:91,2] = PR[GP1:90,2] + 19.320;
   1:L PR[91] R[100]mm/sec CNT100;
   1:  PR[GP1:91,1] = PR[GP1:90,1] + 13.118;
   1:  PR[GP1:91,2] = PR[GP1:90,2] + 19.137;
   1:L PR[91] R[100]mm/sec CNT100;
   1:  PR[GP1:91,1] = PR[GP1:90,1] + 10.704;
   1:  PR[GP1:91,2] = PR[GP1:90,2] + 18.511;
   1:L PR[91] R[100]mm/sec CNT100;
   1:  PR[GP1:91,1] = PR[GP1:90,1] + 8.577;
   1:  PR[GP1:91,2] = PR[GP1:90,2] + 17.581;
   1:L PR[91] R[100]mm/sec CNT100;
   1:  PR[GP1:91,1] = PR[GP1:90,1] + 6.863;
   1:  PR[GP1:91,2] = PR[GP1:90,2] + 16.864;
   1:L PR[91] R[100]mm/sec CNT100;
   1:  PR[GP1:91,1] = PR[GP1:90,1] + 5.059;
   1:  PR[GP1:91,2] = PR[GP1:90,2] + 15.713;
   1:L PR[91] R[100]mm/sec CNT100;
   1:  PR[GP1:91,1] = PR[GP1:90,1] + 4.729;
   1:  PR[GP1:91,2] = PR[GP1:90,2] + 15.485;
   1:L PR[91] R[100]mm/sec CNT100;
   1:  PR[GP1:91,1] = PR[GP1:90,1] + 4.115;
   1:  PR[GP1:91,2] = PR[GP1:90,2] + 14.999;
   1:L PR[91] R[100]mm/sec CNT100;
   1:  PR[GP1:91,1] = PR[GP1:90,1] + 2.650;
   1:  PR[GP1:91,2] = PR[GP1:90,2] + 13.694;
   1:L PR[91] R[100]mm/sec CNT100;
   1:  PR[GP1:91,1] = PR[GP1:90,1] + 2.187;
   1:  PR[GP1:91,2] = PR[GP1:90,2] + 13.207;
   1:L PR[91] R[100]mm/sec CNT100;
   1:  PR[GP1:91,1] = PR[GP1:90,1] + 2.071;
   1:  PR[GP1:91,2] = PR[GP1:90,2] + 13.124;
   1:L PR[91] R[100]mm/sec CNT100;
   1:  PR[GP1:91,1] = PR[GP1:90,1] + 1.975;
   1:  PR[GP1:91,2] = PR[GP1:90,2] + 12.997;
   1:L PR[91] R[100]mm/sec CNT100;
   1:  PR[GP1:91,1] = PR[GP1:90,1] + 1.492;
   1:  PR[GP1:91,2] = PR[GP1:90,2] + 12.655;
   1:L PR[91] R[100]mm/sec CNT100;
   1:  PR[GP1:91,1] = PR[GP1:90,1] + 0.659;
   1:  PR[GP1:91,2] = PR[GP1:90,2] + 12.199;
   1:L PR[91] R[100]mm/sec CNT100;
   1:  PR[GP1:91,1] = PR[GP1:90,1] + -0.537;
   1:L PR[91] R[100]mm/sec CNT100;
   1:  PR[91] = PR[90];
   1:  PR[GP1:91,1] = PR[GP1:90,1] + -1.619;
   1:  PR[GP1:91,2] = PR[GP1:90,2] + 13.007;
   1:  PR[GP1:91,3] = PR[GP1:90,3] + 29.585;
   1:L PR[91] R[100]mm/sec CNT100;
   1:  PR[GP1:91,1] = PR[GP1:90,1] + -2.026;
   1:  PR[GP1:91,2] = PR[GP1:90,2] + 13.535;
   1:L PR[91] R[100]mm/sec CNT100;
   1:  PR[GP1:91,1] = PR[GP1:90,1] + -2.284;
   1:  PR[GP1:91,2] = PR[GP1:90,2] + 13.796;
   1:L PR[91] R[100]mm/sec CNT100;
   1:  PR[GP1:91,1] = PR[GP1:90,1] + -3.663;
   1:  PR[GP1:91,2] = PR[GP1:90,2] + 15.020;
   1:L PR[91] R[100]mm/sec CNT100;
   1:  PR[GP1:91,1] = PR[GP1:90,1] + -4.322;
   1:  PR[GP1:91,2] = PR[GP1:90,2] + 15.541;
   1:L PR[91] R[100]mm/sec CNT100;
   1:  PR[GP1:91,1] = PR[GP1:90,1] + -5.881;
   1:  PR[GP1:91,2] = PR[GP1:90,2] + 16.540;
   1:L PR[91] R[100]mm/sec CNT100;
   1:  PR[GP1:91,1] = PR[GP1:90,1] + -6.447;
   1:  PR[GP1:91,2] = PR[GP1:90,2] + 16.919;
   1:L PR[91] R[100]mm/sec CNT100;
   1:  PR[GP1:91,1] = PR[GP1:90,1] + -8.547;
   1:  PR[GP1:91,2] = PR[GP1:90,2] + 17.837;
   1:L PR[91] R[100]mm/sec CNT100;
   1:  PR[GP1:91,1] = PR[GP1:90,1] + -10.347;
   1:  PR[GP1:91,2] = PR[GP1:90,2] + 18.591;
   1:L PR[91] R[100]mm/sec CNT100;
   1:  PR[GP1:91,1] = PR[GP1:90,1] + -12.616;
   1:  PR[GP1:91,2] = PR[GP1:90,2] + 19.178;
   1:L PR[91] R[100]mm/sec CNT100;
   1:  PR[GP1:91,1] = PR[GP1:90,1] + -15.383;
   1:  PR[GP1:91,2] = PR[GP1:90,2] + 19.466;
   1:L PR[91] R[100]mm/sec CNT100;
   1:  PR[GP1:91,1] = PR[GP1:90,1] + -16.726;
   1:  PR[GP1:91,2] = PR[GP1:90,2] + 19.649;
   1:L PR[91] R[100]mm/sec CNT100;
   1:  PR[GP1:91,1] = PR[GP1:90,1] + -19.525;
   1:  PR[GP1:91,2] = PR[GP1:90,2] + 19.502;
   1:L PR[91] R[100]mm/sec CNT100;
   1:  PR[GP1:91,1] = PR[GP1:90,1] + -20.474;
   1:  PR[GP1:91,2] = PR[GP1:90,2] + 19.389;
   1:L PR[91] R[100]mm/sec CNT100;
   1:  PR[GP1:91,1] = PR[GP1:90,1] + -23.312;
   1:  PR[GP1:91,2] = PR[GP1:90,2] + 18.800;
   1:L PR[91] R[100]mm/sec CNT100;
   1:  PR[GP1:91,1] = PR[GP1:90,1] + -26.695;
   1:  PR[GP1:91,2] = PR[GP1:90,2] + 17.538;
   1:L PR[91] R[100]mm/sec CNT100;
   1:  PR[GP1:91,1] = PR[GP1:90,1] + -29.547;
   1:  PR[GP1:91,2] = PR[GP1:90,2] + 15.940;
   1:L PR[91] R[100]mm/sec CNT100;
   1:  PR[GP1:91,1] = PR[GP1:90,1] + -32.277;
   1:  PR[GP1:91,2] = PR[GP1:90,2] + 13.788;
   1:L PR[91] R[100]mm/sec CNT100;
   1:  PR[GP1:91,1] = PR[GP1:90,1] + -34.179;
   1:  PR[GP1:91,2] = PR[GP1:90,2] + 11.741;
   1:L PR[91] R[100]mm/sec CNT100;
   1:  PR[GP1:91,1] = PR[GP1:90,1] + -34.665;
   1:  PR[GP1:91,2] = PR[GP1:90,2] + 11.063;
   1:L PR[91] R[100]mm/sec CNT100;
   1:  PR[GP1:91,1] = PR[GP1:90,1] + -36.145;
   1:  PR[GP1:91,2] = PR[GP1:90,2] + 8.811;
   1:L PR[91] R[100]mm/sec CNT100;
   1:  PR[GP1:91,1] = PR[GP1:90,1] + -37.114;
   1:  PR[GP1:91,2] = PR[GP1:90,2] + 6.635;
   1:L PR[91] R[100]mm/sec CNT100;
   1:  PR[GP1:91,1] = PR[GP1:90,1] + -37.627;
   1:  PR[GP1:91,2] = PR[GP1:90,2] + 5.357;
   1:L PR[91] R[100]mm/sec CNT100;
   1:  PR[GP1:91,1] = PR[GP1:90,1] + -38.150;
   1:  PR[GP1:91,2] = PR[GP1:90,2] + 3.335;
   1:L PR[91] R[100]mm/sec CNT100;
   1:  PR[GP1:91,1] = PR[GP1:90,1] + -38.352;
   1:  PR[GP1:91,2] = PR[GP1:90,2] + 1.744;
   1:L PR[91] R[100]mm/sec CNT100;
   1:  PR[GP1:91,1] = PR[GP1:90,1] + -38.512;
   1:  PR[GP1:91,2] = PR[GP1:90,2] + -0.277;
   1:L PR[91] R[100]mm/sec CNT100;
   1:  PR[GP1:91,1] = PR[GP1:90,1] + -38.308;
   1:  PR[GP1:91,2] = PR[GP1:90,2] + -1.869;
   1:L PR[91] R[100]mm/sec CNT100;
   1:  PR[GP1:91,1] = PR[GP1:90,1] + -38.141;
   1:  PR[GP1:91,2] = PR[GP1:90,2] + -3.993;
   1:L PR[91] R[100]mm/sec CNT100;
   1:  PR[GP1:91,1] = PR[GP1:90,1] + -37.627;
   1:  PR[GP1:91,2] = PR[GP1:90,2] + -5.981;
   1:L PR[91] R[100]mm/sec CNT100;
   1:  PR[GP1:91,1] = PR[GP1:90,1] + -37.114;
   1:  PR[GP1:91,2] = PR[GP1:90,2] + -7.260;
   1:L PR[91] R[100]mm/sec CNT100;
   1:  PR[GP1:91,1] = PR[GP1:90,1] + -36.157;
   1:  PR[GP1:91,2] = PR[GP1:90,2] + -9.406;
   1:L PR[91] R[100]mm/sec CNT100;
   1:  PR[GP1:91,1] = PR[GP1:90,1] + -35.527;
   1:  PR[GP1:91,2] = PR[GP1:90,2] + -10.281;
   1:L PR[91] R[100]mm/sec CNT100;
   1:  PR[GP1:91,1] = PR[GP1:90,1] + -34.157;
   1:  PR[GP1:91,2] = PR[GP1:90,2] + -12.389;
   1:L PR[91] R[100]mm/sec CNT100;
   1:  PR[GP1:91,1] = PR[GP1:90,1] + -32.259;
   1:  PR[GP1:91,2] = PR[GP1:90,2] + -14.431;
   1:L PR[91] R[100]mm/sec CNT100;
   1:  PR[GP1:91,1] = PR[GP1:90,1] + -32.014;
   1:  PR[GP1:91,2] = PR[GP1:90,2] + -14.638;
   1:L PR[91] R[100]mm/sec CNT100;
   1:  PR[GP1:91,1] = PR[GP1:90,1] + -29.550;
   1:  PR[GP1:91,2] = PR[GP1:90,2] + -16.562;
   1:L PR[91] R[100]mm/sec CNT100;
   1:  PR[GP1:91,1] = PR[GP1:90,1] + -26.695;
   1:  PR[GP1:91,2] = PR[GP1:90,2] + -18.162;
   1:L PR[91] R[100]mm/sec CNT100;
   1:  PR[GP1:91,1] = PR[GP1:90,1] + -23.839;
   1:  PR[GP1:91,2] = PR[GP1:90,2] + -19.216;
   1:L PR[91] R[100]mm/sec CNT100;
   1:  PR[GP1:91,1] = PR[GP1:90,1] + -23.297;
   1:  PR[GP1:91,2] = PR[GP1:90,2] + -19.428;
   1:L PR[91] R[100]mm/sec CNT100;
   1:  PR[GP1:91,1] = PR[GP1:90,1] + -20.469;
   1:  PR[GP1:91,2] = PR[GP1:90,2] + -20.015;
   1:L PR[91] R[100]mm/sec CNT100;
   1:  PR[GP1:91,1] = PR[GP1:90,1] + -19.518;
   1:  PR[GP1:91,2] = PR[GP1:90,2] + -20.125;
   1:L PR[91] R[100]mm/sec CNT100;
   1:  PR[GP1:91,1] = PR[GP1:90,1] + -16.690;
   1:  PR[GP1:91,2] = PR[GP1:90,2] + -20.275;
   1:L PR[91] R[100]mm/sec CNT100;
   1:  PR[GP1:91,1] = PR[GP1:90,1] + -14.178;
   1:  PR[GP1:91,2] = PR[GP1:90,2] + -20.022;
   1:L PR[91] R[100]mm/sec CNT100;
   1:  PR[GP1:91,1] = PR[GP1:90,1] + -12.625;
   1:  PR[GP1:91,2] = PR[GP1:90,2] + -19.804;
   1:L PR[91] R[100]mm/sec CNT100;
   1:  PR[GP1:91,1] = PR[GP1:90,1] + -10.342;
   1:  PR[GP1:91,2] = PR[GP1:90,2] + -19.214;
   1:L PR[91] R[100]mm/sec CNT100;
   1:  PR[GP1:91,1] = PR[GP1:90,1] + -8.326;
   1:  PR[GP1:91,2] = PR[GP1:90,2] + -18.330;
   1:L PR[91] R[100]mm/sec CNT100;
   1:  PR[GP1:91,1] = PR[GP1:90,1] + -6.368;
   1:  PR[GP1:91,2] = PR[GP1:90,2] + -17.495;
   1:L PR[91] R[100]mm/sec CNT100;
   1:  PR[GP1:91,1] = PR[GP1:90,1] + -4.682;
   1:  PR[GP1:91,2] = PR[GP1:90,2] + -16.417;
   1:L PR[91] R[100]mm/sec CNT100;
   1:  PR[GP1:91,1] = PR[GP1:90,1] + -4.107;
   1:  PR[GP1:91,2] = PR[GP1:90,2] + -16.003;
   1:L PR[91] R[100]mm/sec CNT100;
   1:  PR[GP1:91,1] = PR[GP1:90,1] + -2.186;
   1:  PR[GP1:91,2] = PR[GP1:90,2] + -14.321;
   1:L PR[91] R[100]mm/sec CNT100;
   1:  PR[GP1:91,1] = PR[GP1:90,1] + -2.028;
   1:  PR[GP1:91,2] = PR[GP1:90,2] + -14.158;
   1:L PR[91] R[100]mm/sec CNT100;
   1:  PR[GP1:91,1] = PR[GP1:90,1] + -1.445;
   1:  PR[GP1:91,2] = PR[GP1:90,2] + -13.690;
   1:L PR[91] R[100]mm/sec CNT100;
   1:  PR[GP1:91,1] = PR[GP1:90,1] + -0.428;
   1:  PR[GP1:91,2] = PR[GP1:90,2] + -12.971;
   1:L PR[91] R[100]mm/sec CNT100;
   1:  PR[GP1:91,1] = PR[GP1:90,1] + 0.811;
   1:  PR[GP1:91,2] = PR[GP1:90,2] + -13.411;
   1:L PR[91] R[100]mm/sec CNT100;
   1:  PR[GP1:91,1] = PR[GP1:90,1] + 1.263;
   1:L PR[91] R[100]mm/sec CNT100;
   1:  PR[GP1:91,1] = PR[GP1:90,1] + 2.190;
   1:  PR[GP1:91,2] = PR[GP1:90,2] + -14.163;
   1:L PR[91] R[100]mm/sec CNT100;
   1:  PR[GP1:91,1] = PR[GP1:90,1] + 2.348;
   1:  PR[GP1:91,2] = PR[GP1:90,2] + -14.325;
   1:L PR[91] R[100]mm/sec CNT100;
   1:  PR[GP1:91,1] = PR[GP1:90,1] + 4.243;
   1:  PR[GP1:91,2] = PR[GP1:90,2] + -15.987;
   1:L PR[91] R[100]mm/sec CNT100;
   1:  PR[GP1:91,1] = PR[GP1:90,1] + 5.610;
   1:  PR[GP1:91,2] = PR[GP1:90,2] + -16.862;
   1:L PR[91] R[100]mm/sec CNT100;
   1:  PR[GP1:91,1] = PR[GP1:90,1] + 6.547;
   1:  PR[GP1:91,2] = PR[GP1:90,2] + -17.508;
   1:L PR[91] R[100]mm/sec CNT100;
   1:  PR[GP1:91,1] = PR[GP1:90,1] + 10.488;
   1:  PR[GP1:91,2] = PR[GP1:90,2] + -19.209;
   1:L PR[91] R[100]mm/sec CNT100;
   1:  PR[GP1:91,1] = PR[GP1:90,1] + 12.755;
   1:  PR[GP1:91,2] = PR[GP1:90,2] + -19.796;
   1:L PR[91] R[100]mm/sec CNT100;
   1:  PR[GP1:91,1] = PR[GP1:90,1] + 15.518;
   1:  PR[GP1:91,2] = PR[GP1:90,2] + -20.086;
   1:L PR[91] R[100]mm/sec CNT100;
   1:  PR[GP1:91,1] = PR[GP1:90,1] + 16.865;
   1:  PR[GP1:91,2] = PR[GP1:90,2] + -20.273;
   1:L PR[91] R[100]mm/sec CNT100;
   1:  PR[GP1:91,1] = PR[GP1:90,1] + 19.652;
   1:  PR[GP1:91,2] = PR[GP1:90,2] + -20.129;
   1:L PR[91] R[100]mm/sec CNT100;
   1:  PR[GP1:91,1] = PR[GP1:90,1] + 20.605;
   1:  PR[GP1:91,2] = PR[GP1:90,2] + -20.018;
   1:L PR[91] R[100]mm/sec CNT100;
   1:  PR[GP1:91,1] = PR[GP1:90,1] + 23.441;
   1:  PR[GP1:91,2] = PR[GP1:90,2] + -19.431;
   1:L PR[91] R[100]mm/sec CNT100;
   1:  PR[GP1:91,1] = PR[GP1:90,1] + 26.553;
   1:  PR[GP1:91,2] = PR[GP1:90,2] + -18.281;
   1:L PR[91] R[100]mm/sec CNT100;
   1:  PR[GP1:91,1] = PR[GP1:90,1] + 26.823;
   1:  PR[GP1:91,2] = PR[GP1:90,2] + -18.176;
   1:L PR[91] R[100]mm/sec CNT100;
   1:  PR[GP1:91,1] = PR[GP1:90,1] + 29.673;
   1:  PR[GP1:91,2] = PR[GP1:90,2] + -16.588;
   1:L PR[91] R[100]mm/sec CNT100;
   1:  PR[GP1:91,1] = PR[GP1:90,1] + 32.387;
   1:  PR[GP1:91,2] = PR[GP1:90,2] + -14.456;
   1:L PR[91] R[100]mm/sec CNT100;
   1:  PR[GP1:91,1] = PR[GP1:90,1] + 34.304;
   1:  PR[GP1:91,2] = PR[GP1:90,2] + -12.397;
   1:L PR[91] R[100]mm/sec CNT100;
   1:  PR[GP1:91,1] = PR[GP1:90,1] + 34.787;
   1:  PR[GP1:91,2] = PR[GP1:90,2] + -11.722;
   1:L PR[91] R[100]mm/sec CNT100;
   1:  PR[GP1:91,1] = PR[GP1:90,1] + 36.293;
   1:  PR[GP1:91,2] = PR[GP1:90,2] + -9.444;
   1:L PR[91] R[100]mm/sec CNT100;
   1:  PR[GP1:91,1] = PR[GP1:90,1] + 37.261;
   1:  PR[GP1:91,2] = PR[GP1:90,2] + -7.300;
   1:L PR[91] R[100]mm/sec CNT100;
   1:  PR[GP1:91,1] = PR[GP1:90,1] + 37.773;
   1:  PR[GP1:91,2] = PR[GP1:90,2] + -6.031;
   1:L PR[91] R[100]mm/sec CNT100;
   1:  PR[GP1:91,1] = PR[GP1:90,1] + 38.297;
   1:  PR[GP1:91,2] = PR[GP1:90,2] + -4.030;
   1:L PR[91] R[100]mm/sec CNT100;
   1:  PR[GP1:91,1] = PR[GP1:90,1] + 38.499;
   1:  PR[GP1:91,2] = PR[GP1:90,2] + -2.435;
   1:L PR[91] R[100]mm/sec CNT100;
   1:  PR[GP1:91,1] = PR[GP1:90,1] + 38.668;
   1:  PR[GP1:91,2] = PR[GP1:90,2] + -0.345;
   1:L PR[91] R[100]mm/sec CNT100;
   1:  PR[GP1:91,1] = PR[GP1:90,1] + 38.465;
   1:  PR[GP1:91,2] = PR[GP1:90,2] + 1.250;
   1:L PR[91] R[100]mm/sec CNT100;
   1:  PR[GP1:91,1] = PR[GP1:90,1] + 38.289;
   1:  PR[GP1:91,2] = PR[GP1:90,2] + 3.439;
   1:L PR[91] R[100]mm/sec CNT100;
   1:  PR[GP1:91,1] = PR[GP1:90,1] + 37.773;
   1:  PR[GP1:91,2] = PR[GP1:90,2] + 5.408;
   1:L PR[91] R[100]mm/sec CNT100;
   1:  PR[GP1:91,1] = PR[GP1:90,1] + 37.260;
   1:  PR[GP1:91,2] = PR[GP1:90,2] + 6.676;
   1:L PR[91] R[100]mm/sec CNT100;
   1:  PR[GP1:91,1] = PR[GP1:90,1] + 36.304;
   1:  PR[GP1:91,2] = PR[GP1:90,2] + 8.794;
   1:L PR[91] R[100]mm/sec CNT100;
   1:  PR[GP1:91,1] = PR[GP1:90,1] + 35.674;
   1:  PR[GP1:91,2] = PR[GP1:90,2] + 9.669;
   1:L PR[91] R[100]mm/sec CNT100;
   1:  PR[GP1:91,1] = PR[GP1:90,1] + 34.283;
   1:  PR[GP1:91,2] = PR[GP1:90,2] + 11.796;
   1:L PR[91] R[100]mm/sec CNT100;
   1:  PR[GP1:91,1] = PR[GP1:90,1] + 32.368;
   1:  PR[GP1:91,2] = PR[GP1:90,2] + 13.853;
   1:L PR[91] R[100]mm/sec CNT100;
   1:  PR[GP1:91,1] = PR[GP1:90,1] + 32.130;
   1:  PR[GP1:91,2] = PR[GP1:90,2] + 14.055;
   1:L PR[91] R[100]mm/sec CNT100;
   1:  PR[GP1:91,1] = PR[GP1:90,1] + 29.677;
   1:  PR[GP1:91,2] = PR[GP1:90,2] + 15.962;
   1:L PR[91] R[100]mm/sec CNT100;
   1:  PR[GP1:91,1] = PR[GP1:90,1] + 26.836;
   1:  PR[GP1:91,2] = PR[GP1:90,2] + 17.544;
   1:L PR[91] R[100]mm/sec CNT100;
   1:  PR[GP1:91,1] = PR[GP1:90,1] + 23.975;
   1:  PR[GP1:91,2] = PR[GP1:90,2] + 18.596;
   1:L PR[91] R[100]mm/sec CNT100;
   1:  PR[GP1:91,1] = PR[GP1:90,1] + 23.432;
   1:  PR[GP1:91,2] = PR[GP1:90,2] + 18.808;
   1:L PR[91] R[100]mm/sec CNT100;
   1:  PR[GP1:91,1] = PR[GP1:90,1] + 20.609;
   1:  PR[GP1:91,2] = PR[GP1:90,2] + 19.392;
   1:L PR[91] R[100]mm/sec CNT100;
   1:  PR[GP1:91,1] = PR[GP1:90,1] + 19.659;
   1:  PR[GP1:91,2] = PR[GP1:90,2] + 19.505;
   1:L PR[91] R[100]mm/sec CNT100;
   1:  PR[GP1:91,1] = PR[GP1:90,1] + 16.849;
   1:  PR[GP1:91,2] = PR[GP1:90,2] + 19.651;
   1:L PR[91] R[100]mm/sec CNT100;
   1:  PR[GP1:91,1] = PR[GP1:90,1] + 14.343;
   1:  PR[GP1:91,2] = PR[GP1:90,2] + 19.397;
   1:L PR[91] R[100]mm/sec CNT100;
   1:  PR[GP1:91,1] = PR[GP1:90,1] + 12.793;
   1:  PR[GP1:91,2] = PR[GP1:90,2] + 19.182;
   1:L PR[91] R[100]mm/sec CNT100;
   1:  PR[GP1:91,1] = PR[GP1:90,1] + 10.508;
   1:  PR[GP1:91,2] = PR[GP1:90,2] + 18.590;
   1:L PR[91] R[100]mm/sec CNT100;
   1:  PR[GP1:91,1] = PR[GP1:90,1] + 8.492;
   1:  PR[GP1:91,2] = PR[GP1:90,2] + 17.708;
   1:L PR[91] R[100]mm/sec CNT100;
   1:  PR[GP1:91,1] = PR[GP1:90,1] + 6.576;
   1:  PR[GP1:91,2] = PR[GP1:90,2] + 16.907;
   1:L PR[91] R[100]mm/sec CNT100;
   1:  PR[GP1:91,1] = PR[GP1:90,1] + 4.877;
   1:  PR[GP1:91,2] = PR[GP1:90,2] + 15.823;
   1:L PR[91] R[100]mm/sec CNT100;
   1:  PR[GP1:91,1] = PR[GP1:90,1] + 4.508;
   1:  PR[GP1:91,2] = PR[GP1:90,2] + 15.568;
   1:L PR[91] R[100]mm/sec CNT100;
   1:  PR[GP1:91,1] = PR[GP1:90,1] + 3.827;
   1:  PR[GP1:91,2] = PR[GP1:90,2] + 15.029;
   1:L PR[91] R[100]mm/sec CNT100;
   1:  PR[GP1:91,1] = PR[GP1:90,1] + 2.455;
   1:  PR[GP1:91,2] = PR[GP1:90,2] + 13.810;
   1:L PR[91] R[100]mm/sec CNT100;
   1:  PR[GP1:91,1] = PR[GP1:90,1] + 2.167;
   1:  PR[GP1:91,2] = PR[GP1:90,2] + 13.507;
   1:L PR[91] R[100]mm/sec CNT100;
   1:  PR[GP1:91,1] = PR[GP1:90,1] + 1.982;
   1:  PR[GP1:91,2] = PR[GP1:90,2] + 13.374;
   1:L PR[91] R[100]mm/sec CNT100;
   1:  PR[GP1:91,1] = PR[GP1:90,1] + 1.918;
   1:  PR[GP1:91,2] = PR[GP1:90,2] + 13.290;
   1:L PR[91] R[100]mm/sec CNT100;
   1:  PR[GP1:91,1] = PR[GP1:90,1] + 1.516;
   1:  PR[GP1:91,2] = PR[GP1:90,2] + 13.005;
   1:L PR[91] R[100]mm/sec CNT100;
   1:  PR[GP1:91,1] = PR[GP1:90,1] + 0.619;
   1:  PR[GP1:91,2] = PR[GP1:90,2] + 12.514;
   1:L PR[91] R[100]mm/sec CNT100;
   1:  PR[GP1:91,1] = PR[GP1:90,1] + -0.513;
   1:L PR[91] R[100]mm/sec CNT100;
   1:  PR[91] = PR[90];
   1:  PR[GP1:91,1] = PR[GP1:90,1] + -1.659;
   1:  PR[GP1:91,2] = PR[GP1:90,2] + 13.350;
   1:  PR[GP1:91,3] = PR[GP1:90,3] + 30.195;
   1:L PR[91] R[100]mm/sec CNT100;
   1:  PR[GP1:91,1] = PR[GP1:90,1] + -2.094;
   1:  PR[GP1:91,2] = PR[GP1:90,2] + 13.916;
   1:L PR[91] R[100]mm/sec CNT100;
   1:  PR[GP1:91,1] = PR[GP1:90,1] + -3.375;
   1:  PR[GP1:91,2] = PR[GP1:90,2] + 15.051;
   1:L PR[91] R[100]mm/sec CNT100;
   1:  PR[GP1:91,1] = PR[GP1:90,1] + -4.102;
   1:  PR[GP1:91,2] = PR[GP1:90,2] + 15.625;
   1:L PR[91] R[100]mm/sec CNT100;
   1:  PR[GP1:91,1] = PR[GP1:90,1] + -5.528;
   1:  PR[GP1:91,2] = PR[GP1:90,2] + 16.538;
   1:L PR[91] R[100]mm/sec CNT100;
   1:  PR[GP1:91,1] = PR[GP1:90,1] + -6.160;
   1:  PR[GP1:91,2] = PR[GP1:90,2] + 16.962;
   1:L PR[91] R[100]mm/sec CNT100;
   1:  PR[GP1:91,1] = PR[GP1:90,1] + -8.132;
   1:  PR[GP1:91,2] = PR[GP1:90,2] + 17.824;
   1:L PR[91] R[100]mm/sec CNT100;
   1:  PR[GP1:91,1] = PR[GP1:90,1] + -10.152;
   1:  PR[GP1:91,2] = PR[GP1:90,2] + 18.670;
   1:L PR[91] R[100]mm/sec CNT100;
   1:  PR[GP1:91,1] = PR[GP1:90,1] + -12.291;
   1:  PR[GP1:91,2] = PR[GP1:90,2] + 19.223;
   1:L PR[91] R[100]mm/sec CNT100;
   1:  PR[GP1:91,1] = PR[GP1:90,1] + -14.909;
   1:  PR[GP1:91,2] = PR[GP1:90,2] + 19.496;
   1:L PR[91] R[100]mm/sec CNT100;
   1:  PR[GP1:91,1] = PR[GP1:90,1] + -16.502;
   1:  PR[GP1:91,2] = PR[GP1:90,2] + 19.713;
   1:L PR[91] R[100]mm/sec CNT100;
   1:  PR[GP1:91,1] = PR[GP1:90,1] + -19.158;
   1:  PR[GP1:91,2] = PR[GP1:90,2] + 19.573;
   1:L PR[91] R[100]mm/sec CNT100;
   1:  PR[GP1:91,1] = PR[GP1:90,1] + -20.349;
   1:  PR[GP1:91,2] = PR[GP1:90,2] + 19.432;
   1:L PR[91] R[100]mm/sec CNT100;
   1:  PR[GP1:91,1] = PR[GP1:90,1] + -23.053;
   1:  PR[GP1:91,2] = PR[GP1:90,2] + 18.871;
   1:L PR[91] R[100]mm/sec CNT100;
   1:  PR[GP1:91,1] = PR[GP1:90,1] + -26.533;
   1:  PR[GP1:91,2] = PR[GP1:90,2] + 17.568;
   1:L PR[91] R[100]mm/sec CNT100;
   1:  PR[GP1:91,1] = PR[GP1:90,1] + -29.264;
   1:  PR[GP1:91,2] = PR[GP1:90,2] + 16.038;
   1:L PR[91] R[100]mm/sec CNT100;
   1:  PR[GP1:91,1] = PR[GP1:90,1] + -31.985;
   1:  PR[GP1:91,2] = PR[GP1:90,2] + 13.921;
   1:L PR[91] R[100]mm/sec CNT100;
   1:  PR[GP1:91,1] = PR[GP1:90,1] + -34.103;
   1:  PR[GP1:91,2] = PR[GP1:90,2] + 11.641;
   1:L PR[91] R[100]mm/sec CNT100;
   1:  PR[GP1:91,1] = PR[GP1:90,1] + -34.288;
   1:  PR[GP1:91,2] = PR[GP1:90,2] + 11.383;
   1:L PR[91] R[100]mm/sec CNT100;
   1:  PR[GP1:91,1] = PR[GP1:90,1] + -35.967;
   1:  PR[GP1:91,2] = PR[GP1:90,2] + 8.828;
   1:L PR[91] R[100]mm/sec CNT100;
   1:  PR[GP1:91,1] = PR[GP1:90,1] + -37.068;
   1:  PR[GP1:91,2] = PR[GP1:90,2] + 6.358;
   1:L PR[91] R[100]mm/sec CNT100;
   1:  PR[GP1:91,1] = PR[GP1:90,1] + -37.409;
   1:  PR[GP1:91,2] = PR[GP1:90,2] + 5.507;
   1:L PR[91] R[100]mm/sec CNT100;
   1:  PR[GP1:91,1] = PR[GP1:90,1] + -38.011;
   1:  PR[GP1:91,2] = PR[GP1:90,2] + 3.181;
   1:L PR[91] R[100]mm/sec CNT100;
   1:  PR[GP1:91,1] = PR[GP1:90,1] + -38.152;
   1:  PR[GP1:91,2] = PR[GP1:90,2] + 2.067;
   1:L PR[91] R[100]mm/sec CNT100;
   1:  PR[GP1:91,1] = PR[GP1:90,1] + -38.338;
   1:  PR[GP1:91,2] = PR[GP1:90,2] + -0.277;
   1:L PR[91] R[100]mm/sec CNT100;
   1:  PR[GP1:91,1] = PR[GP1:90,1] + -38.193;
   1:  PR[GP1:91,2] = PR[GP1:90,2] + -1.409;
   1:L PR[91] R[100]mm/sec CNT100;
   1:  PR[GP1:91,1] = PR[GP1:90,1] + -38.002;
   1:  PR[GP1:91,2] = PR[GP1:90,2] + -3.839;
   1:L PR[91] R[100]mm/sec CNT100;
   1:  PR[GP1:91,1] = PR[GP1:90,1] + -37.409;
   1:  PR[GP1:91,2] = PR[GP1:90,2] + -6.131;
   1:L PR[91] R[100]mm/sec CNT100;
   1:  PR[GP1:91,1] = PR[GP1:90,1] + -37.068;
   1:  PR[GP1:91,2] = PR[GP1:90,2] + -6.982;
   1:L PR[91] R[100]mm/sec CNT100;
   1:  PR[GP1:91,1] = PR[GP1:90,1] + -35.980;
   1:  PR[GP1:91,2] = PR[GP1:90,2] + -9.423;
   1:L PR[91] R[100]mm/sec CNT100;
   1:  PR[GP1:91,1] = PR[GP1:90,1] + -35.613;
   1:  PR[GP1:91,2] = PR[GP1:90,2] + -9.933;
   1:L PR[91] R[100]mm/sec CNT100;
   1:  PR[GP1:91,1] = PR[GP1:90,1] + -34.081;
   1:  PR[GP1:91,2] = PR[GP1:90,2] + -12.289;
   1:L PR[91] R[100]mm/sec CNT100;
   1:  PR[GP1:91,1] = PR[GP1:90,1] + -31.984;
   1:  PR[GP1:91,2] = PR[GP1:90,2] + -14.547;
   1:L PR[91] R[100]mm/sec CNT100;
   1:  PR[GP1:91,1] = PR[GP1:90,1] + -29.447;
   1:  PR[GP1:91,2] = PR[GP1:90,2] + -16.533;
   1:L PR[91] R[100]mm/sec CNT100;
   1:  PR[GP1:91,1] = PR[GP1:90,1] + -29.283;
   1:  PR[GP1:91,2] = PR[GP1:90,2] + -16.651;
   1:L PR[91] R[100]mm/sec CNT100;
   1:  PR[GP1:91,1] = PR[GP1:90,1] + -26.533;
   1:  PR[GP1:91,2] = PR[GP1:90,2] + -18.192;
   1:L PR[91] R[100]mm/sec CNT100;
   1:  PR[GP1:91,1] = PR[GP1:90,1] + -23.799;
   1:  PR[GP1:91,2] = PR[GP1:90,2] + -19.202;
   1:L PR[91] R[100]mm/sec CNT100;
   1:  PR[GP1:91,1] = PR[GP1:90,1] + -23.037;
   1:  PR[GP1:91,2] = PR[GP1:90,2] + -19.499;
   1:L PR[91] R[100]mm/sec CNT100;
   1:  PR[GP1:91,1] = PR[GP1:90,1] + -20.342;
   1:  PR[GP1:91,2] = PR[GP1:90,2] + -20.058;
   1:L PR[91] R[100]mm/sec CNT100;
   1:  PR[GP1:91,1] = PR[GP1:90,1] + -19.149;
   1:  PR[GP1:91,2] = PR[GP1:90,2] + -20.197;
   1:L PR[91] R[100]mm/sec CNT100;
   1:  PR[GP1:91,1] = PR[GP1:90,1] + -16.464;
   1:  PR[GP1:91,2] = PR[GP1:90,2] + -20.339;
   1:L PR[91] R[100]mm/sec CNT100;
   1:  PR[GP1:91,1] = PR[GP1:90,1] + -14.079;
   1:  PR[GP1:91,2] = PR[GP1:90,2] + -20.098;
   1:L PR[91] R[100]mm/sec CNT100;
   1:  PR[GP1:91,1] = PR[GP1:90,1] + -12.298;
   1:  PR[GP1:91,2] = PR[GP1:90,2] + -19.849;
   1:L PR[91] R[100]mm/sec CNT100;
   1:  PR[GP1:91,1] = PR[GP1:90,1] + -10.145;
   1:  PR[GP1:91,2] = PR[GP1:90,2] + -19.292;
   1:L PR[91] R[100]mm/sec CNT100;
   1:  PR[GP1:91,1] = PR[GP1:90,1] + -8.239;
   1:  PR[GP1:91,2] = PR[GP1:90,2] + -18.456;
   1:L PR[91] R[100]mm/sec CNT100;
   1:  PR[GP1:91,1] = PR[GP1:90,1] + -6.075;
   1:  PR[GP1:91,2] = PR[GP1:90,2] + -17.534;
   1:L PR[91] R[100]mm/sec CNT100;
   1:  PR[GP1:91,1] = PR[GP1:90,1] + -4.497;
   1:  PR[GP1:91,2] = PR[GP1:90,2] + -16.525;
   1:L PR[91] R[100]mm/sec CNT100;
   1:  PR[GP1:91,1] = PR[GP1:90,1] + -3.863;
   1:  PR[GP1:91,2] = PR[GP1:90,2] + -16.068;
   1:L PR[91] R[100]mm/sec CNT100;
   1:  PR[GP1:91,1] = PR[GP1:90,1] + -1.774;
   1:  PR[GP1:91,2] = PR[GP1:90,2] + -14.239;
   1:L PR[91] R[100]mm/sec CNT100;
   1:  PR[GP1:91,1] = PR[GP1:90,1] + -1.656;
   1:  PR[GP1:91,2] = PR[GP1:90,2] + -14.199;
   1:L PR[91] R[100]mm/sec CNT100;
   1:  PR[GP1:91,1] = PR[GP1:90,1] + -1.368;
   1:  PR[GP1:91,2] = PR[GP1:90,2] + -13.968;
   1:L PR[91] R[100]mm/sec CNT100;
   1:  PR[GP1:91,1] = PR[GP1:90,1] + -0.403;
   1:  PR[GP1:91,2] = PR[GP1:90,2] + -13.286;
   1:L PR[91] R[100]mm/sec CNT100;
   1:  PR[GP1:91,1] = PR[GP1:90,1] + 0.934;
   1:  PR[GP1:91,2] = PR[GP1:90,2] + -13.761;
   1:L PR[91] R[100]mm/sec CNT100;
   1:  PR[GP1:91,1] = PR[GP1:90,1] + 1.291;
   1:L PR[91] R[100]mm/sec CNT100;
   1:  PR[GP1:91,1] = PR[GP1:90,1] + 1.872;
   1:  PR[GP1:91,2] = PR[GP1:90,2] + -14.236;
   1:L PR[91] R[100]mm/sec CNT100;
   1:  PR[GP1:91,1] = PR[GP1:90,1] + 2.053;
   1:  PR[GP1:91,2] = PR[GP1:90,2] + -14.346;
   1:L PR[91] R[100]mm/sec CNT100;
   1:  PR[GP1:91,1] = PR[GP1:90,1] + 3.998;
   1:  PR[GP1:91,2] = PR[GP1:90,2] + -16.051;
   1:L PR[91] R[100]mm/sec CNT100;
   1:  PR[GP1:91,1] = PR[GP1:90,1] + 5.213;
   1:  PR[GP1:91,2] = PR[GP1:90,2] + -16.830;
   1:L PR[91] R[100]mm/sec CNT100;
   1:  PR[GP1:91,1] = PR[GP1:90,1] + 6.256;
   1:  PR[GP1:91,2] = PR[GP1:90,2] + -17.548;
   1:L PR[91] R[100]mm/sec CNT100;
   1:  PR[GP1:91,1] = PR[GP1:90,1] + 8.196;
   1:  PR[GP1:91,2] = PR[GP1:90,2] + -18.395;
   1:L PR[91] R[100]mm/sec CNT100;
   1:  PR[GP1:91,1] = PR[GP1:90,1] + 10.288;
   1:  PR[GP1:91,2] = PR[GP1:90,2] + -19.286;
   1:L PR[91] R[100]mm/sec CNT100;
   1:  PR[GP1:91,1] = PR[GP1:90,1] + 12.428;
   1:  PR[GP1:91,2] = PR[GP1:90,2] + -19.841;
   1:L PR[91] R[100]mm/sec CNT100;
   1:  PR[GP1:91,1] = PR[GP1:90,1] + 15.043;
   1:  PR[GP1:91,2] = PR[GP1:90,2] + -20.115;
   1:L PR[91] R[100]mm/sec CNT100;
   1:  PR[GP1:91,1] = PR[GP1:90,1] + 16.640;
   1:  PR[GP1:91,2] = PR[GP1:90,2] + -20.337;
   1:L PR[91] R[100]mm/sec CNT100;
   1:  PR[GP1:91,1] = PR[GP1:90,1] + 19.284;
   1:  PR[GP1:91,2] = PR[GP1:90,2] + -20.200;
   1:L PR[91] R[100]mm/sec CNT100;
   1:  PR[GP1:91,1] = PR[GP1:90,1] + 20.479;
   1:  PR[GP1:91,2] = PR[GP1:90,2] + -20.061;
   1:L PR[91] R[100]mm/sec CNT100;
   1:  PR[GP1:91,1] = PR[GP1:90,1] + 23.182;
   1:  PR[GP1:91,2] = PR[GP1:90,2] + -19.501;
   1:L PR[91] R[100]mm/sec CNT100;
   1:  PR[GP1:91,1] = PR[GP1:90,1] + 26.151;
   1:  PR[GP1:91,2] = PR[GP1:90,2] + -18.405;
   1:L PR[91] R[100]mm/sec CNT100;
   1:  PR[GP1:91,1] = PR[GP1:90,1] + 26.661;
   1:  PR[GP1:91,2] = PR[GP1:90,2] + -18.206;
   1:L PR[91] R[100]mm/sec CNT100;
   1:  PR[GP1:91,1] = PR[GP1:90,1] + 29.390;
   1:  PR[GP1:91,2] = PR[GP1:90,2] + -16.686;
   1:L PR[91] R[100]mm/sec CNT100;
   1:  PR[GP1:91,1] = PR[GP1:90,1] + 32.093;
   1:  PR[GP1:91,2] = PR[GP1:90,2] + -14.592;
   1:L PR[91] R[100]mm/sec CNT100;
   1:  PR[GP1:91,1] = PR[GP1:90,1] + 34.224;
   1:  PR[GP1:91,2] = PR[GP1:90,2] + -12.301;
   1:L PR[91] R[100]mm/sec CNT100;
   1:  PR[GP1:91,1] = PR[GP1:90,1] + 34.406;
   1:  PR[GP1:91,2] = PR[GP1:90,2] + -12.048;
   1:L PR[91] R[100]mm/sec CNT100;
   1:  PR[GP1:91,1] = PR[GP1:90,1] + 36.114;
   1:  PR[GP1:91,2] = PR[GP1:90,2] + -9.464;
   1:L PR[91] R[100]mm/sec CNT100;
   1:  PR[GP1:91,1] = PR[GP1:90,1] + 37.213;
   1:  PR[GP1:91,2] = PR[GP1:90,2] + -7.029;
   1:L PR[91] R[100]mm/sec CNT100;
   1:  PR[GP1:91,1] = PR[GP1:90,1] + 37.553;
   1:  PR[GP1:91,2] = PR[GP1:90,2] + -6.186;
   1:L PR[91] R[100]mm/sec CNT100;
   1:  PR[GP1:91,1] = PR[GP1:90,1] + 38.157;
   1:  PR[GP1:91,2] = PR[GP1:90,2] + -3.884;
   1:L PR[91] R[100]mm/sec CNT100;
   1:  PR[GP1:91,1] = PR[GP1:90,1] + 38.298;
   1:  PR[GP1:91,2] = PR[GP1:90,2] + -2.768;
   1:L PR[91] R[100]mm/sec CNT100;
   1:  PR[GP1:91,1] = PR[GP1:90,1] + 38.494;
   1:  PR[GP1:91,2] = PR[GP1:90,2] + -0.345;
   1:L PR[91] R[100]mm/sec CNT100;
   1:  PR[GP1:91,1] = PR[GP1:90,1] + 38.350;
   1:  PR[GP1:91,2] = PR[GP1:90,2] + 0.789;
   1:L PR[91] R[100]mm/sec CNT100;
   1:  PR[GP1:91,1] = PR[GP1:90,1] + 38.148;
   1:  PR[GP1:91,2] = PR[GP1:90,2] + 3.292;
   1:L PR[91] R[100]mm/sec CNT100;
   1:  PR[GP1:91,1] = PR[GP1:90,1] + 37.553;
   1:  PR[GP1:91,2] = PR[GP1:90,2] + 5.562;
   1:L PR[91] R[100]mm/sec CNT100;
   1:  PR[GP1:91,1] = PR[GP1:90,1] + 37.213;
   1:  PR[GP1:91,2] = PR[GP1:90,2] + 6.405;
   1:L PR[91] R[100]mm/sec CNT100;
   1:  PR[GP1:91,1] = PR[GP1:90,1] + 36.126;
   1:  PR[GP1:91,2] = PR[GP1:90,2] + 8.814;
   1:L PR[91] R[100]mm/sec CNT100;
   1:  PR[GP1:91,1] = PR[GP1:90,1] + 35.759;
   1:  PR[GP1:91,2] = PR[GP1:90,2] + 9.323;
   1:L PR[91] R[100]mm/sec CNT100;
   1:  PR[GP1:91,1] = PR[GP1:90,1] + 34.203;
   1:  PR[GP1:91,2] = PR[GP1:90,2] + 11.700;
   1:L PR[91] R[100]mm/sec CNT100;
   1:  PR[GP1:91,1] = PR[GP1:90,1] + 32.093;
   1:  PR[GP1:91,2] = PR[GP1:90,2] + 13.968;
   1:L PR[91] R[100]mm/sec CNT100;
   1:  PR[GP1:91,1] = PR[GP1:90,1] + 29.391;
   1:  PR[GP1:91,2] = PR[GP1:90,2] + 16.061;
   1:L PR[91] R[100]mm/sec CNT100;
   1:  PR[GP1:91,1] = PR[GP1:90,1] + 26.675;
   1:  PR[GP1:91,2] = PR[GP1:90,2] + 17.574;
   1:L PR[91] R[100]mm/sec CNT100;
   1:  PR[GP1:91,1] = PR[GP1:90,1] + 23.937;
   1:  PR[GP1:91,2] = PR[GP1:90,2] + 18.580;
   1:L PR[91] R[100]mm/sec CNT100;
   1:  PR[GP1:91,1] = PR[GP1:90,1] + 23.175;
   1:  PR[GP1:91,2] = PR[GP1:90,2] + 18.879;
   1:L PR[91] R[100]mm/sec CNT100;
   1:  PR[GP1:91,1] = PR[GP1:90,1] + 20.485;
   1:  PR[GP1:91,2] = PR[GP1:90,2] + 19.435;
   1:L PR[91] R[100]mm/sec CNT100;
   1:  PR[GP1:91,1] = PR[GP1:90,1] + 19.293;
   1:  PR[GP1:91,2] = PR[GP1:90,2] + 19.576;
   1:L PR[91] R[100]mm/sec CNT100;
   1:  PR[GP1:91,1] = PR[GP1:90,1] + 16.625;
   1:  PR[GP1:91,2] = PR[GP1:90,2] + 19.715;
   1:L PR[91] R[100]mm/sec CNT100;
   1:  PR[GP1:91,1] = PR[GP1:90,1] + 14.246;
   1:  PR[GP1:91,2] = PR[GP1:90,2] + 19.474;
   1:L PR[91] R[100]mm/sec CNT100;
   1:  PR[GP1:91,1] = PR[GP1:90,1] + 12.468;
   1:  PR[GP1:91,2] = PR[GP1:90,2] + 19.228;
   1:L PR[91] R[100]mm/sec CNT100;
   1:  PR[GP1:91,1] = PR[GP1:90,1] + 10.313;
   1:  PR[GP1:91,2] = PR[GP1:90,2] + 18.669;
   1:L PR[91] R[100]mm/sec CNT100;
   1:  PR[GP1:91,1] = PR[GP1:90,1] + 8.406;
   1:  PR[GP1:91,2] = PR[GP1:90,2] + 17.835;
   1:L PR[91] R[100]mm/sec CNT100;
   1:  PR[GP1:91,1] = PR[GP1:90,1] + 6.288;
   1:  PR[GP1:91,2] = PR[GP1:90,2] + 16.950;
   1:L PR[91] R[100]mm/sec CNT100;
   1:  PR[GP1:91,1] = PR[GP1:90,1] + 4.694;
   1:  PR[GP1:91,2] = PR[GP1:90,2] + 15.932;
   1:L PR[91] R[100]mm/sec CNT100;
   1:  PR[GP1:91,1] = PR[GP1:90,1] + 4.288;
   1:  PR[GP1:91,2] = PR[GP1:90,2] + 15.651;
   1:L PR[91] R[100]mm/sec CNT100;
   1:  PR[GP1:91,1] = PR[GP1:90,1] + 3.541;
   1:  PR[GP1:91,2] = PR[GP1:90,2] + 15.060;
   1:L PR[91] R[100]mm/sec CNT100;
   1:  PR[GP1:91,1] = PR[GP1:90,1] + 2.114;
   1:  PR[GP1:91,2] = PR[GP1:90,2] + 13.785;
   1:L PR[91] R[100]mm/sec CNT100;
   1:  PR[GP1:91,1] = PR[GP1:90,1] + 1.561;
   1:  PR[GP1:91,2] = PR[GP1:90,2] + 13.366;
   1:L PR[91] R[100]mm/sec CNT100;
   1:  PR[GP1:91,1] = PR[GP1:90,1] + 0.579;
   1:  PR[GP1:91,2] = PR[GP1:90,2] + 12.829;
   1:L PR[91] R[100]mm/sec CNT100;
   1:  PR[GP1:91,1] = PR[GP1:90,1] + -0.489;
   1:L PR[91] R[100]mm/sec CNT100;
   1:  PR[91] = PR[90];
   1:  PR[GP1:91,1] = PR[GP1:90,1] + -1.698;
   1:  PR[GP1:91,2] = PR[GP1:90,2] + 13.693;
   1:  PR[GP1:91,3] = PR[GP1:90,3] + 30.805;
   1:L PR[91] R[100]mm/sec CNT100;
   1:  PR[GP1:91,1] = PR[GP1:90,1] + -2.079;
   1:  PR[GP1:91,2] = PR[GP1:90,2] + 14.189;
   1:L PR[91] R[100]mm/sec CNT100;
   1:  PR[GP1:91,1] = PR[GP1:90,1] + -3.089;
   1:  PR[GP1:91,2] = PR[GP1:90,2] + 15.082;
   1:L PR[91] R[100]mm/sec CNT100;
   1:  PR[GP1:91,1] = PR[GP1:90,1] + -3.882;
   1:  PR[GP1:91,2] = PR[GP1:90,2] + 15.709;
   1:L PR[91] R[100]mm/sec CNT100;
   1:  PR[GP1:91,1] = PR[GP1:90,1] + -5.175;
   1:  PR[GP1:91,2] = PR[GP1:90,2] + 16.537;
   1:L PR[91] R[100]mm/sec CNT100;
   1:  PR[GP1:91,1] = PR[GP1:90,1] + -5.873;
   1:  PR[GP1:91,2] = PR[GP1:90,2] + 17.005;
   1:L PR[91] R[100]mm/sec CNT100;
   1:  PR[GP1:91,1] = PR[GP1:90,1] + -7.717;
   1:  PR[GP1:91,2] = PR[GP1:90,2] + 17.811;
   1:L PR[91] R[100]mm/sec CNT100;
   1:  PR[GP1:91,1] = PR[GP1:90,1] + -9.956;
   1:  PR[GP1:91,2] = PR[GP1:90,2] + 18.749;
   1:L PR[91] R[100]mm/sec CNT100;
   1:  PR[GP1:91,1] = PR[GP1:90,1] + -11.966;
   1:  PR[GP1:91,2] = PR[GP1:90,2] + 19.269;
   1:L PR[91] R[100]mm/sec CNT100;
   1:  PR[GP1:91,1] = PR[GP1:90,1] + -14.435;
   1:  PR[GP1:91,2] = PR[GP1:90,2] + 19.526;
   1:L PR[91] R[100]mm/sec CNT100;
   1:  PR[GP1:91,1] = PR[GP1:90,1] + -16.278;
   1:  PR[GP1:91,2] = PR[GP1:90,2] + 19.777;
   1:L PR[91] R[100]mm/sec CNT100;
   1:  PR[GP1:91,1] = PR[GP1:90,1] + -18.791;
   1:  PR[GP1:91,2] = PR[GP1:90,2] + 19.645;
   1:L PR[91] R[100]mm/sec CNT100;
   1:  PR[GP1:91,1] = PR[GP1:90,1] + -20.224;
   1:  PR[GP1:91,2] = PR[GP1:90,2] + 19.475;
   1:L PR[91] R[100]mm/sec CNT100;
   1:  PR[GP1:91,1] = PR[GP1:90,1] + -22.797;
   1:  PR[GP1:91,2] = PR[GP1:90,2] + 18.941;
   1:L PR[91] R[100]mm/sec CNT100;
   1:  PR[GP1:91,1] = PR[GP1:90,1] + -25.617;
   1:  PR[GP1:91,2] = PR[GP1:90,2] + 17.895;
   1:L PR[91] R[100]mm/sec CNT100;
   1:  PR[GP1:91,1] = PR[GP1:90,1] + -26.362;
   1:  PR[GP1:91,2] = PR[GP1:90,2] + 17.603;
   1:L PR[91] R[100]mm/sec CNT100;
   1:  PR[GP1:91,1] = PR[GP1:90,1] + -28.977;
   1:  PR[GP1:91,2] = PR[GP1:90,2] + 16.138;
   1:L PR[91] R[100]mm/sec CNT100;
   1:  PR[GP1:91,1] = PR[GP1:90,1] + -31.789;
   1:  PR[GP1:91,2] = PR[GP1:90,2] + 13.961;
   1:L PR[91] R[100]mm/sec CNT100;
   1:  PR[GP1:91,1] = PR[GP1:90,1] + -33.974;
   1:  PR[GP1:91,2] = PR[GP1:90,2] + 11.601;
   1:L PR[91] R[100]mm/sec CNT100;
   1:  PR[GP1:91,1] = PR[GP1:90,1] + -35.790;
   1:  PR[GP1:91,2] = PR[GP1:90,2] + 8.844;
   1:L PR[91] R[100]mm/sec CNT100;
   1:  PR[GP1:91,1] = PR[GP1:90,1] + -37.022;
   1:  PR[GP1:91,2] = PR[GP1:90,2] + 6.081;
   1:L PR[91] R[100]mm/sec CNT100;
   1:  PR[GP1:91,1] = PR[GP1:90,1] + -37.192;
   1:  PR[GP1:91,2] = PR[GP1:90,2] + 5.657;
   1:L PR[91] R[100]mm/sec CNT100;
   1:  PR[GP1:91,1] = PR[GP1:90,1] + -37.872;
   1:  PR[GP1:91,2] = PR[GP1:90,2] + 3.028;
   1:L PR[91] R[100]mm/sec CNT100;
   1:  PR[GP1:91,1] = PR[GP1:90,1] + -37.953;
   1:  PR[GP1:91,2] = PR[GP1:90,2] + 2.390;
   1:L PR[91] R[100]mm/sec CNT100;
   1:  PR[GP1:91,1] = PR[GP1:90,1] + -38.164;
   1:  PR[GP1:91,2] = PR[GP1:90,2] + -0.277;
   1:L PR[91] R[100]mm/sec CNT100;
   1:  PR[GP1:91,1] = PR[GP1:90,1] + -38.078;
   1:  PR[GP1:91,2] = PR[GP1:90,2] + -0.950;
   1:L PR[91] R[100]mm/sec CNT100;
   1:  PR[GP1:91,1] = PR[GP1:90,1] + -37.863;
   1:  PR[GP1:91,2] = PR[GP1:90,2] + -3.685;
   1:L PR[91] R[100]mm/sec CNT100;
   1:  PR[GP1:91,1] = PR[GP1:90,1] + -37.192;
   1:  PR[GP1:91,2] = PR[GP1:90,2] + -6.281;
   1:L PR[91] R[100]mm/sec CNT100;
   1:  PR[GP1:91,1] = PR[GP1:90,1] + -37.022;
   1:  PR[GP1:91,2] = PR[GP1:90,2] + -6.705;
   1:L PR[91] R[100]mm/sec CNT100;
   1:  PR[GP1:91,1] = PR[GP1:90,1] + -35.803;
   1:  PR[GP1:91,2] = PR[GP1:90,2] + -9.440;
   1:L PR[91] R[100]mm/sec CNT100;
   1:  PR[GP1:91,1] = PR[GP1:90,1] + -35.699;
   1:  PR[GP1:91,2] = PR[GP1:90,2] + -9.584;
   1:L PR[91] R[100]mm/sec CNT100;
   1:  PR[GP1:91,1] = PR[GP1:90,1] + -33.995;
   1:  PR[GP1:91,2] = PR[GP1:90,2] + -12.198;
   1:L PR[91] R[100]mm/sec CNT100;
   1:  PR[GP1:91,1] = PR[GP1:90,1] + -31.785;
   1:  PR[GP1:91,2] = PR[GP1:90,2] + -14.589;
   1:L PR[91] R[100]mm/sec CNT100;
   1:  PR[GP1:91,1] = PR[GP1:90,1] + -29.358;
   1:  PR[GP1:91,2] = PR[GP1:90,2] + -16.489;
   1:L PR[91] R[100]mm/sec CNT100;
   1:  PR[GP1:91,1] = PR[GP1:90,1] + -28.995;
   1:  PR[GP1:91,2] = PR[GP1:90,2] + -16.752;
   1:L PR[91] R[100]mm/sec CNT100;
   1:  PR[GP1:91,1] = PR[GP1:90,1] + -26.370;
   1:  PR[GP1:91,2] = PR[GP1:90,2] + -18.223;
   1:L PR[91] R[100]mm/sec CNT100;
   1:  PR[GP1:91,1] = PR[GP1:90,1] + -23.758;
   1:  PR[GP1:91,2] = PR[GP1:90,2] + -19.187;
   1:L PR[91] R[100]mm/sec CNT100;
   1:  PR[GP1:91,1] = PR[GP1:90,1] + -22.778;
   1:  PR[GP1:91,2] = PR[GP1:90,2] + -19.570;
   1:L PR[91] R[100]mm/sec CNT100;
   1:  PR[GP1:91,1] = PR[GP1:90,1] + -20.216;
   1:  PR[GP1:91,2] = PR[GP1:90,2] + -20.101;
   1:L PR[91] R[100]mm/sec CNT100;
   1:  PR[GP1:91,1] = PR[GP1:90,1] + -18.779;
   1:  PR[GP1:91,2] = PR[GP1:90,2] + -20.269;
   1:L PR[91] R[100]mm/sec CNT100;
   1:  PR[GP1:91,1] = PR[GP1:90,1] + -16.238;
   1:  PR[GP1:91,2] = PR[GP1:90,2] + -20.403;
   1:L PR[91] R[100]mm/sec CNT100;
   1:  PR[GP1:91,1] = PR[GP1:90,1] + -13.980;
   1:  PR[GP1:91,2] = PR[GP1:90,2] + -20.175;
   1:L PR[91] R[100]mm/sec CNT100;
   1:  PR[GP1:91,1] = PR[GP1:90,1] + -11.971;
   1:  PR[GP1:91,2] = PR[GP1:90,2] + -19.894;
   1:L PR[91] R[100]mm/sec CNT100;
   1:  PR[GP1:91,1] = PR[GP1:90,1] + -9.947;
   1:  PR[GP1:91,2] = PR[GP1:90,2] + -19.371;
   1:L PR[91] R[100]mm/sec CNT100;
   1:  PR[GP1:91,1] = PR[GP1:90,1] + -8.151;
   1:  PR[GP1:91,2] = PR[GP1:90,2] + -18.583;
   1:L PR[91] R[100]mm/sec CNT100;
   1:  PR[GP1:91,1] = PR[GP1:90,1] + -5.782;
   1:  PR[GP1:91,2] = PR[GP1:90,2] + -17.573;
   1:L PR[91] R[100]mm/sec CNT100;
   1:  PR[GP1:91,1] = PR[GP1:90,1] + -4.312;
   1:  PR[GP1:91,2] = PR[GP1:90,2] + -16.634;
   1:L PR[91] R[100]mm/sec CNT100;
   1:  PR[GP1:91,1] = PR[GP1:90,1] + -3.619;
   1:  PR[GP1:91,2] = PR[GP1:90,2] + -16.134;
   1:L PR[91] R[100]mm/sec CNT100;
   1:  PR[GP1:91,1] = PR[GP1:90,1] + -1.756;
